C05457=1013.009,-114.708,391.527,-28.818,50.485,-33.096
C05458=1013.004,-115.096,391.557,-28.834,50.637,-33.068
C05459=1013.000,-115.485,391.587,-28.849,50.788,-33.043
C05460=1012.996,-115.873,391.617,-28.865,50.941,-33.016
C05461=1012.993,-116.261,391.647,-28.881,51.094,-32.989
C05462=1012.990,-116.650,391.676,-28.897,51.248,-32.964
C05463=1012.985,-117.038,391.706,-28.913,51.403,-32.938
C05464=1012.982,-117.427,391.737,-28.928,51.558,-32.911
C05465=1012.978,-117.814,391.766,-28.944,51.713,-32.886
C05466=1012.974,-118.203,391.796,-28.960,51.870,-32.860
C05467=1012.970,-118.591,391.826,-28.977,52.028,-32.834
C05468=1012.966,-118.979,391.856,-28.993,52.187,-32.809
C05469=1012.962,-119.367,391.886,-29.009,52.345,-32.783
C05470=1012.959,-119.756,391.916,-29.025,52.504,-32.759
C05471=1012.955,-120.143,391.945,-29.042,52.665,-32.734
C05472=1012.951,-120.532,391.976,-29.058,52.825,-32.709
C05473=1012.947,-120.920,392.005,-29.075,52.986,-32.685
C05474=1012.943,-121.308,392.035,-29.091,53.148,-32.660
C05475=1012.939,-121.696,392.065,-29.108,53.311,-32.636
C05476=1012.936,-122.084,392.095,-29.125,53.475,-32.612
C05477=1012.932,-122.472,392.125,-29.141,53.639,-32.587
C05478=1012.928,-122.861,392.155,-29.158,53.804,-32.564
C05479=1012.924,-123.248,392.184,-29.176,53.969,-32.541
C05480=1012.920,-123.637,392.215,-29.193,54.135,-32.518
C05481=1012.917,-124.025,392.244,-29.210,54.303,-32.495
C05482=1012.913,-124.413,392.274,-29.227,54.470,-32.472
C05483=1012.909,-124.800,392.304,-29.244,54.638,-32.449
C05484=1012.905,-125.188,392.334,-29.262,54.807,-32.427
C05485=1012.901,-125.577,392.364,-29.280,54.977,-32.405
C05486=1012.898,-125.964,392.394,-29.297,55.147,-32.383
C05487=1012.894,-126.352,392.424,-29.315,55.317,-32.362
C05488=1012.890,-126.741,392.454,-29.333,55.489,-32.340
C05489=1012.886,-127.128,392.484,-29.351,55.662,-32.319
C05490=1012.883,-127.516,392.514,-29.369,55.833,-32.297
C05491=1012.878,-127.904,392.544,-29.388,56.007,-32.278
C05492=1012.875,-128.292,392.574,-29.406,56.181,-32.258
C05493=1012.871,-128.679,392.604,-29.424,56.355,-32.238
C05494=1012.867,-129.067,392.634,-29.443,56.531,-32.217
C05495=1012.863,-129.455,392.664,-29.462,56.707,-32.197
C05496=1012.860,-129.843,392.694,-29.481,56.884,-32.179
C05497=1012.855,-130.231,392.724,-29.500,57.062,-32.160
C05498=1012.852,-130.619,392.754,-29.519,57.238,-32.142
C05499=1012.848,-131.006,392.784,-29.538,57.418,-32.123
C05500=1012.845,-131.394,392.814,-29.558,57.597,-32.106
C05501=1012.840,-131.782,392.844,-29.578,57.777,-32.088
C05502=1012.837,-132.170,392.874,-29.597,57.956,-32.071
C05503=1012.833,-132.558,392.903,-29.618,58.138,-32.054
C05504=1012.830,-132.945,392.934,-29.637,58.320,-32.037
C05505=1012.825,-133.333,392.964,-29.658,58.502,-32.021
C05506=1012.822,-133.721,392.994,-29.678,58.685,-32.005
C05507=1012.818,-134.108,393.024,-29.699,58.868,-31.991
C05508=1013.072,-134.133,392.609,-28.595,48.020,-33.821
C05509=1013.077,-133.746,392.579,-28.574,47.825,-33.863
C05510=1013.082,-133.358,392.550,-28.553,47.631,-33.906
C05511=1013.087,-132.970,392.521,-28.532,47.438,-33.948
C05512=1013.092,-132.582,392.491,-28.511,47.244,-33.991
C05513=1013.097,-132.194,392.461,-28.490,47.051,-34.034
C05514=1013.103,-131.806,392.431,-28.469,46.860,-34.077
C05515=1013.108,-131.418,392.402,-28.448,46.669,-34.121
C05516=1013.113,-131.031,392.372,-28.427,46.479,-34.165
C05517=1013.118,-130.643,392.343,-28.406,46.290,-34.208
C05518=1013.122,-130.255,392.314,-28.384,46.101,-34.254
C05519=1013.127,-129.868,392.283,-28.363,45.913,-34.297
C05520=1013.132,-129.480,392.254,-28.342,45.725,-34.342
C05521=1013.138,-129.092,392.225,-28.321,45.538,-34.387
C05522=1013.143,-128.704,392.195,-28.300,45.352,-34.432
C05523=1013.148,-128.316,392.165,-28.279,45.168,-34.477
C05524=1013.153,-127.928,392.136,-28.257,44.983,-34.524
C05525=1013.158,-127.540,392.107,-28.236,44.799,-34.569
C05526=1013.164,-127.152,392.077,-28.215,44.616,-34.614
C05527=1013.168,-126.764,392.047,-28.193,44.434,-34.660
C05528=1013.173,-126.376,392.018,-28.172,44.252,-34.706
C05529=1013.179,-125.988,391.989,-28.151,44.071,-34.753
C05530=1013.183,-125.600,391.959,-28.130,43.891,-34.799
C05531=1013.189,-125.212,391.929,-28.108,43.712,-34.846
C05532=1013.193,-124.825,391.901,-28.087,43.533,-34.893
C05533=1013.199,-124.437,391.871,-28.065,43.355,-34.940
C05534=1013.203,-124.049,391.842,-28.044,43.178,-34.987
C05535=1013.208,-123.661,391.813,-28.023,43.001,-35.034
C05536=1013.214,-123.273,391.783,-28.001,42.826,-35.082
C05537=1013.218,-122.885,391.753,-27.980,42.651,-35.129
C05538=1013.223,-122.497,391.724,-27.958,42.478,-35.176
C05539=1013.229,-122.109,391.695,-27.937,42.304,-35.225
C05540=1013.233,-121.721,391.665,-27.915,42.131,-35.273
C05541=1013.238,-121.333,391.636,-27.894,41.959,-35.320
C05542=1013.244,-120.945,391.606,-27.872,41.788,-35.369
C05543=1013.248,-120.556,391.577,-27.850,41.617,-35.417
C05544=1013.253,-120.168,391.548,-27.829,41.448,-35.464
C05545=1013.259,-119.780,391.518,-27.807,41.280,-35.512
C05546=1013.263,-119.392,391.489,-27.786,41.112,-35.561
C05547=1013.268,-119.004,391.459,-27.764,40.944,-35.610
C05548=1013.274,-118.616,391.430,-27.742,40.778,-35.658
C05549=1013.278,-118.227,391.400,-27.721,40.612,-35.707
C05550=1013.283,-117.839,391.371,-27.699,40.447,-35.756
C05551=1013.287,-117.450,391.342,-27.677,40.283,-35.805
C05552=1013.293,-117.062,391.313,-27.655,40.119,-35.854
C05553=1013.298,-116.674,391.284,-27.634,39.957,-35.902
C05554=1013.302,-116.286,391.254,-27.612,39.795,-35.953
C05555=1013.308,-115.897,391.225,-27.590,39.634,-36.001
C05556=1013.312,-115.508,391.196,-27.568,39.474,-36.051
C05557=1013.318,-115.120,391.166,-27.547,39.314,-36.099
C05558=1013.322,-114.732,391.137,-27.525,39.155,-36.149
C05559=1013.327,-114.344,391.108,-27.503,38.997,-36.198
C05560=1013.332,-113.955,391.078,-27.481,38.840,-36.247
C05561=1013.336,-113.597,391.052,-27.461,38.696,-36.293
C05562=1013.341,-113.179,391.020,-27.438,38.529,-36.346
C05563=1013.346,-112.790,390.991,-27.416,38.374,-36.395
C05564=1013.351,-112.402,390.961,-27.394,38.220,-36.445
C05565=1013.355,-112.013,390.932,-27.372,38.067,-36.494
C05566=1013.361,-111.624,390.903,-27.350,37.914,-36.543
C05567=1013.365,-111.235,390.874,-27.328,37.763,-36.593
C05568=1013.370,-110.847,390.845,-27.306,37.612,-36.642
C05569=1013.374,-110.458,390.815,-27.285,37.462,-36.693
C05570=1013.379,-110.070,390.786,-27.263,37.313,-36.741
C05571=1013.384,-109.681,390.757,-27.241,37.165,-36.790
C05572=1013.389,-109.287,390.727,-27.219,37.015,-36.841
C05573=1013.393,-108.870,390.695,-27.195,36.859,-36.892
C05574=1013.395,-108.651,390.679,-27.183,36.776,-36.921
C05575=1013.398,-108.426,390.662,-27.170,36.692,-36.949
C05576=1013.401,-108.196,390.645,-27.157,36.606,-36.979
C05577=1013.404,-107.964,390.627,-27.144,36.521,-37.008
C05578=1013.406,-107.732,390.610,-27.131,36.434,-37.038
C05579=1013.409,-107.502,390.593,-27.118,36.349,-37.068
C05580=1013.413,-107.275,390.576,-27.105,36.265,-37.097
C05581=1013.414,-107.055,390.560,-27.093,36.184,-37.125
C05582=1013.417,-106.841,390.544,-27.081,36.106,-37.152
C05583=1013.422,-106.434,390.512,-27.058,35.958,-37.202
C05584=1013.426,-106.044,390.483,-27.036,35.816,-37.252
C05585=1013.431,-105.655,390.454,-27.015,35.676,-37.300
C05586=1013.435,-105.266,390.425,-26.993,35.537,-37.350
C05587=1013.440,-104.878,390.396,-26.971,35.400,-37.398
C05588=1013.444,-104.490,390.366,-26.949,35.263,-37.447
C05589=1013.448,-104.103,390.338,-26.928,35.127,-37.495
C05590=1013.453,-103.716,390.309,-26.906,34.992,-37.544
C05591=1013.457,-103.330,390.280,-26.885,34.859,-37.592
C05592=1013.462,-102.944,390.250,-26.863,34.726,-37.640
C05593=1013.465,-102.558,390.222,-26.842,34.594,-37.687
C05594=1013.470,-102.174,390.193,-26.821,34.463,-37.736
C05595=1013.474,-101.791,390.164,-26.799,34.334,-37.783
C05596=1013.478,-101.408,390.135,-26.778,34.205,-37.830
C05597=1013.482,-101.026,390.106,-26.757,34.078,-37.877
C05598=1013.487,-100.645,390.078,-26.736,33.951,-37.924
C05599=1013.491,-100.266,390.049,-26.715,33.826,-37.971
C05600=1013.495,-99.888,390.021,-26.694,33.703,-38.017
C05601=1013.498,-99.510,389.993,-26.674,33.580,-38.063
C05602=1013.502,-99.133,389.965,-26.653,33.459,-38.109
C05603=1013.507,-98.758,389.937,-26.633,33.338,-38.155
C05604=1013.511,-98.381,389.908,-26.612,33.218,-38.200
C05605=1013.515,-98.006,389.880,-26.592,33.100,-38.244
C05606=1013.519,-97.632,389.852,-26.572,32.982,-38.290
C05607=1013.522,-97.256,389.824,-26.551,32.865,-38.335
C05608=1013.526,-96.879,389.795,-26.531,32.749,-38.378
C05609=1013.530,-96.503,389.768,-26.511,32.634,-38.423
C05610=1013.535,-96.126,389.739,-26.491,32.519,-38.467
C05611=1013.538,-95.748,389.711,-26.471,32.404,-38.512
C05612=1013.541,-95.368,389.683,-26.450,32.291,-38.556
C05613=1013.545,-94.988,389.654,-26.430,32.178,-38.600
C05614=1013.549,-94.606,389.625,-26.410,32.065,-38.644
C05615=1013.553,-94.223,389.597,-26.390,31.952,-38.689
C05616=1013.557,-93.840,389.568,-26.370,31.842,-38.733
C05617=1013.561,-93.455,389.539,-26.350,31.730,-38.778
C05618=1013.564,-93.069,389.510,-26.329,31.619,-38.822
C05619=1013.568,-92.682,389.481,-26.310,31.510,-38.865
C05620=1013.572,-92.295,389.452,-26.290,31.401,-38.909
C05621=1013.576,-91.907,389.423,-26.269,31.292,-38.952
C05622=1013.579,-91.519,389.394,-26.249,31.184,-38.996
C05623=1013.583,-91.130,389.364,-26.230,31.077,-39.039
C05624=1013.586,-90.775,389.338,-26.212,30.980,-39.080
C05625=1013.588,-90.507,389.318,-26.198,30.907,-39.108
C05626=1013.591,-90.296,389.302,-26.187,30.850,-39.131
C05627=1013.593,-90.062,389.285,-26.176,30.788,-39.157
C05628=1013.594,-89.812,389.266,-26.163,30.721,-39.183
C05629=1013.597,-89.553,389.246,-26.150,30.652,-39.212
C05630=1013.599,-89.297,389.227,-26.137,30.585,-39.240
C05631=1013.602,-89.055,389.209,-26.125,30.522,-39.266
C05632=1013.603,-88.836,389.193,-26.114,30.464,-39.289
C05633=1013.607,-88.451,389.164,-26.095,30.364,-39.331
C05634=1013.610,-88.074,389.136,-26.077,30.268,-39.370
C05635=1013.614,-87.712,389.109,-26.059,30.175,-39.409
C05636=1013.617,-87.344,389.080,-26.041,30.082,-39.448
C05637=1013.620,-86.968,389.052,-26.023,29.988,-39.486
C05638=1013.623,-86.579,389.024,-26.004,29.891,-39.527
C05639=1013.627,-86.173,388.993,-25.984,29.791,-39.568
C05640=1013.629,-85.949,388.977,-25.974,29.737,-39.591
C05641=1013.631,-85.715,388.958,-25.963,29.679,-39.614
C05642=1013.633,-85.476,388.940,-25.951,29.622,-39.639
C05643=1013.634,-85.237,388.922,-25.940,29.564,-39.663
C05644=1013.637,-85.008,388.905,-25.929,29.510,-39.686
C05645=1013.640,-84.589,388.875,-25.910,29.411,-39.728
C05646=1013.643,-84.197,388.845,-25.891,29.319,-39.766
C05647=1013.646,-83.806,388.815,-25.873,29.228,-39.805
C05648=1013.650,-83.410,388.785,-25.855,29.137,-39.844
C05649=1013.653,-83.013,388.756,-25.837,29.047,-39.882
C05650=1013.656,-82.618,388.726,-25.819,28.957,-39.920
C05651=1013.660,-82.220,388.696,-25.801,28.869,-39.957
C05652=1013.662,-81.821,388.666,-25.783,28.780,-39.996
C05653=1013.665,-81.423,388.636,-25.765,28.694,-40.032
C05654=1013.668,-81.027,388.607,-25.748,28.608,-40.069
C05655=1013.672,-80.629,388.577,-25.731,28.524,-40.105
C05656=1013.674,-80.231,388.547,-25.713,28.439,-40.142
C05657=1013.677,-79.831,388.516,-25.696,28.356,-40.177
C05658=1013.680,-79.431,388.487,-25.679,28.273,-40.214
C05659=1013.683,-79.031,388.456,-25.662,28.192,-40.248
C05660=1013.686,-78.630,388.426,-25.645,28.110,-40.284
C05661=1013.689,-78.228,388.396,-25.629,28.030,-40.318
C05662=1013.692,-77.828,388.366,-25.612,27.951,-40.352
C05663=1013.694,-77.426,388.336,-25.596,27.873,-40.386
C05664=1013.697,-77.024,388.305,-25.579,27.795,-40.421
C05665=1013.700,-76.622,388.275,-25.563,27.718,-40.454
C05666=1013.703,-76.219,388.245,-25.547,27.643,-40.486
C05667=1013.705,-75.817,388.214,-25.531,27.568,-40.519
C05668=1013.708,-75.414,388.183,-25.516,27.493,-40.552
C05669=1013.710,-75.011,388.154,-25.500,27.420,-40.584
C05670=1013.714,-74.608,388.123,-25.485,27.349,-40.615
C05671=1013.715,-74.205,388.093,-25.469,27.277,-40.646
C05672=1013.718,-73.801,388.062,-25.454,27.206,-40.675
C05673=1013.721,-73.398,388.032,-25.440,27.137,-40.706
C05674=1013.723,-72.994,388.001,-25.425,27.068,-40.737
C05675=1013.725,-72.590,387.971,-25.410,27.000,-40.766
C05676=1013.728,-72.186,387.940,-25.396,26.934,-40.795
C05677=1013.731,-71.783,387.910,-25.381,26.868,-40.823
C05678=1013.733,-71.379,387.880,-25.367,26.804,-40.852
C05679=1013.735,-70.975,387.849,-25.353,26.739,-40.879
C05680=1013.737,-70.571,387.818,-25.340,26.676,-40.908
C05681=1013.739,-70.167,387.788,-25.326,26.614,-40.934
C05682=1013.742,-69.762,387.757,-25.313,26.552,-40.961
C05683=1013.744,-69.358,387.727,-25.300,26.492,-40.986
C05684=1013.746,-68.954,387.697,-25.286,26.432,-41.013
C05685=1013.747,-68.549,387.666,-25.274,26.375,-41.038
C05686=1013.750,-68.145,387.636,-25.261,26.316,-41.064
C05687=1013.752,-67.741,387.605,-25.248,26.259,-41.087
C05688=1013.754,-67.338,387.575,-25.236,26.204,-41.111
C05689=1013.755,-66.933,387.544,-25.224,26.149,-41.136
C05690=1013.758,-66.530,387.512,-25.212,26.095,-41.159
C05691=1013.760,-66.127,387.482,-25.200,26.042,-41.180
C05692=1013.762,-65.723,387.452,-25.189,25.990,-41.203
C05693=1013.764,-65.320,387.421,-25.177,25.938,-41.225
C05694=1013.765,-64.918,387.391,-25.166,25.888,-41.247
C05695=1013.767,-64.516,387.360,-25.155,25.839,-41.268
C05696=1013.768,-64.114,387.329,-25.144,25.791,-41.288
C05697=1013.770,-63.712,387.300,-25.134,25.744,-41.308
C05698=1013.772,-63.311,387.269,-25.123,25.697,-41.328
C05699=1013.774,-62.911,387.238,-25.113,25.651,-41.347
C05700=1013.775,-62.510,387.208,-25.103,25.607,-41.366
C05701=1013.777,-62.110,387.177,-25.094,25.563,-41.384
C05702=1013.778,-61.711,387.147,-25.084,25.520,-41.401
C05703=1013.780,-61.312,387.116,-25.075,25.478,-41.418
C05704=1013.782,-60.914,387.086,-25.066,25.437,-41.435
C05705=1013.783,-60.515,387.056,-25.057,25.397,-41.452
C05706=1013.784,-60.119,387.026,-25.048,25.358,-41.467
C05707=1013.786,-59.722,386.996,-25.039,25.320,-41.483
C05708=1013.787,-59.327,386.966,-25.031,25.282,-41.497
C05709=1013.789,-58.930,386.936,-25.023,25.246,-41.512
C05710=1013.790,-58.535,386.906,-25.015,25.211,-41.525
C05711=1013.791,-58.140,386.875,-25.007,25.176,-41.539
C05712=1013.792,-57.746,386.845,-25.000,25.143,-41.552
C05713=1013.794,-57.353,386.815,-24.993,25.110,-41.564
C05714=1013.794,-56.959,386.785,-24.986,25.078,-41.577
C05715=1013.795,-56.566,386.755,-24.979,25.046,-41.587
C05716=1013.796,-56.173,386.725,-24.972,25.016,-41.598
C05717=1013.797,-55.781,386.695,-24.966,24.987,-41.610
C05718=1013.798,-55.388,386.665,-24.959,24.958,-41.620
C05719=1013.799,-54.996,386.635,-24.953,24.931,-41.631
C05720=1013.800,-54.603,386.605,-24.947,24.904,-41.640
C05721=1013.802,-54.211,386.575,-24.942,24.878,-41.647
C05722=1013.802,-53.818,386.545,-24.936,24.853,-41.656
C05723=1013.803,-53.427,386.515,-24.931,24.828,-41.664
C05724=1013.804,-53.034,386.486,-24.926,24.805,-41.672
C05725=1013.804,-52.641,386.455,-24.921,24.781,-41.679
C05726=1013.805,-52.248,386.425,-24.916,24.760,-41.686
C05727=1013.807,-51.856,386.395,-24.912,24.738,-41.693
C05728=1013.807,-51.464,386.366,-24.907,24.718,-41.698
C05729=1013.807,-51.072,386.335,-24.903,24.698,-41.704
C05730=1013.808,-50.679,386.305,-24.899,24.679,-41.708
C05731=1013.809,-50.287,386.275,-24.896,24.662,-41.712
C05732=1013.810,-49.893,386.244,-24.892,24.644,-41.717
C05733=1013.810,-49.501,386.215,-24.889,24.628,-41.720
C05734=1013.810,-49.109,386.184,-24.885,24.612,-41.723
C05735=1013.811,-48.716,386.154,-24.883,24.598,-41.725
C05736=1013.812,-48.324,386.123,-24.880,24.584,-41.728
C05737=1013.811,-47.931,386.094,-24.877,24.571,-41.729
C05738=1013.812,-47.538,386.064,-24.875,24.558,-41.731
C05739=1013.813,-47.146,386.033,-24.873,24.547,-41.731
C05740=1013.813,-46.753,386.003,-24.871,24.536,-41.732
C05741=1013.813,-46.361,385.973,-24.869,24.525,-41.732
C05742=1013.814,-45.968,385.942,-24.867,24.517,-41.731
C05743=1013.814,-45.575,385.912,-24.866,24.508,-41.731
C05744=1013.814,-45.182,385.882,-24.865,24.501,-41.729
C05745=1013.814,-44.789,385.852,-24.864,24.494,-41.727
C05746=1013.814,-44.397,385.821,-24.863,24.489,-41.724
C05747=1013.814,-44.004,385.791,-24.863,24.483,-41.721
C05748=1013.814,-43.611,385.761,-24.862,24.479,-41.719
C05749=1013.814,-43.217,385.730,-24.862,24.475,-41.715
C05750=1013.815,-42.824,385.700,-24.862,24.473,-41.711
C05751=1013.815,-42.431,385.670,-24.862,24.471,-41.706
C05752=1013.814,-42.039,385.640,-24.863,24.469,-41.702
C05753=1013.814,-41.645,385.609,-24.863,24.469,-41.696
C05754=1013.814,-41.253,385.578,-24.864,24.469,-41.690
C05755=1013.814,-40.860,385.548,-24.865,24.471,-41.684
C05756=1013.815,-40.466,385.518,-24.866,24.473,-41.677
C05757=1013.814,-40.073,385.487,-24.868,24.476,-41.670
C05758=1013.814,-39.680,385.457,-24.869,24.479,-41.663
C05759=1013.813,-39.287,385.426,-24.871,24.483,-41.654
C05760=1013.813,-38.894,385.396,-24.873,24.489,-41.645
C05761=1013.813,-38.501,385.365,-24.875,24.495,-41.637
C05762=1013.812,-38.107,385.336,-24.878,24.501,-41.626
C05763=1013.812,-37.713,385.305,-24.880,24.509,-41.618
C05764=1013.812,-37.320,385.275,-24.883,24.518,-41.606
C05765=1013.811,-36.927,385.244,-24.886,24.526,-41.596
C05766=1013.811,-36.533,385.213,-24.889,24.536,-41.586
C05767=1013.810,-36.141,385.182,-24.892,24.547,-41.574
C05768=1013.810,-35.747,385.152,-24.896,24.558,-41.562
C05769=1013.809,-35.354,385.121,-24.899,24.570,-41.550
C05770=1013.809,-34.961,385.090,-24.903,24.583,-41.537
C05771=1013.808,-34.567,385.060,-24.907,24.596,-41.523
C05772=1013.807,-34.174,385.029,-24.912,24.611,-41.509
C05773=1013.807,-33.781,385.000,-24.916,24.626,-41.496
C05774=1013.806,-33.387,384.969,-24.921,24.643,-41.481
C05775=1013.806,-32.994,384.938,-24.925,24.659,-41.466
C05776=1013.804,-32.601,384.908,-24.930,24.676,-41.451
C05777=1013.804,-32.207,384.877,-24.935,24.695,-41.435
C05778=1013.803,-31.814,384.846,-24.941,24.714,-41.419
C05779=1013.802,-31.420,384.814,-24.946,24.734,-41.402
C05780=1013.800,-31.027,384.785,-24.952,24.755,-41.385
C05781=1013.800,-30.633,384.754,-24.958,24.776,-41.367
C05782=1013.799,-30.240,384.723,-24.964,24.798,-41.350
C05783=1013.798,-29.847,384.693,-24.970,24.821,-41.332
C05784=1013.797,-29.454,384.662,-24.977,24.845,-41.313
C05785=1013.796,-29.061,384.631,-24.983,24.869,-41.294
C05786=1013.795,-28.667,384.600,-24.990,24.894,-41.274
C05787=1013.794,-28.275,384.569,-24.996,24.920,-41.255
C05788=1013.793,-27.880,384.539,-25.004,24.947,-41.234
C05789=1013.791,-27.487,384.508,-25.011,24.975,-41.214
C05790=1013.790,-27.094,384.477,-25.018,25.003,-41.193
C05791=1013.789,-26.701,384.447,-25.026,25.032,-41.171
C05792=1013.788,-26.307,384.415,-25.034,25.062,-41.149
C05793=1013.787,-25.915,384.385,-25.041,25.092,-41.128
C05794=1013.786,-25.522,384.354,-25.050,25.123,-41.105
C05795=1013.784,-25.128,384.323,-25.058,25.155,-41.082
C05796=1013.783,-24.735,384.293,-25.066,25.188,-41.058
C05797=1013.781,-24.342,384.261,-25.075,25.222,-41.035
C05798=1013.781,-23.949,384.231,-25.083,25.255,-41.010
C05799=1013.779,-23.556,384.200,-25.092,25.291,-40.986
C05800=1013.777,-23.163,384.168,-25.101,25.327,-40.962
C05801=1013.775,-22.770,384.139,-25.110,25.363,-40.937
C05802=1013.774,-22.376,384.107,-25.120,25.400,-40.912
C05803=1013.773,-21.983,384.077,-25.129,25.438,-40.885
C05804=1013.771,-21.590,384.046,-25.139,25.477,-40.859
C05805=1013.769,-21.197,384.015,-25.149,25.517,-40.832
C05806=1013.768,-20.804,383.984,-25.159,25.557,-40.805
C05807=1013.766,-20.407,383.953,-25.169,25.598,-40.777
C05808=1013.764,-20.058,383.925,-25.178,25.635,-40.753
C05809=1013.763,-19.852,383.909,-25.183,25.657,-40.738
C05810=1013.762,-19.621,383.891,-25.189,25.683,-40.721
C05811=1013.761,-19.365,383.871,-25.196,25.711,-40.702
C05812=1013.760,-19.091,383.849,-25.204,25.741,-40.683
C05813=1013.759,-18.812,383.828,-25.211,25.772,-40.663
C05814=1013.757,-18.540,383.805,-25.219,25.803,-40.642
C05815=1013.757,-18.287,383.786,-25.226,25.832,-40.623
C05816=1013.756,-18.060,383.768,-25.232,25.858,-40.607
C05817=1013.753,-17.664,383.737,-25.243,25.905,-40.577
C05818=1013.751,-17.275,383.706,-25.254,25.951,-40.547
C05819=1013.749,-16.877,383.674,-25.266,26.000,-40.516
C05820=1013.747,-16.481,383.643,-25.278,26.049,-40.485
C05821=1013.745,-16.085,383.612,-25.289,26.098,-40.454
C05822=1013.744,-15.690,383.581,-25.301,26.148,-40.423
C05823=1013.742,-15.303,383.551,-25.312,26.197,-40.392
C05824=1013.739,-14.923,383.520,-25.324,26.248,-40.360
C05825=1013.737,-14.548,383.491,-25.336,26.296,-40.329
C05826=1013.735,-14.173,383.461,-25.348,26.348,-40.297
C05827=1013.733,-13.792,383.431,-25.360,26.399,-40.264
C05828=1013.732,-13.399,383.400,-25.372,26.453,-40.232
C05829=1013.729,-12.995,383.368,-25.385,26.510,-40.198
C05830=1013.726,-12.584,383.336,-25.398,26.568,-40.162
C05831=1013.724,-12.170,383.303,-25.412,26.627,-40.126
C05832=1013.722,-11.755,383.271,-25.426,26.688,-40.089
C05833=1013.719,-11.337,383.238,-25.440,26.750,-40.052
C05834=1013.717,-10.919,383.204,-25.454,26.812,-40.014
C05835=1013.714,-10.500,383.171,-25.468,26.876,-39.977
C05836=1013.712,-10.080,383.138,-25.483,26.940,-39.938
C05837=1013.709,-9.658,383.105,-25.497,27.005,-39.900
C05838=1013.707,-9.236,383.071,-25.512,27.072,-39.860
C05839=1013.704,-8.814,383.038,-25.527,27.139,-39.821
C05840=1013.702,-8.603,383.021,-25.534,27.173,-39.800
C05841=1013.701,-8.392,383.004,-25.542,27.207,-39.781
C05842=1013.699,-8.034,382.976,-25.555,27.266,-39.747
C05843=1013.696,-7.755,382.954,-25.565,27.311,-39.721
C05844=1013.696,-7.541,382.937,-25.572,27.347,-39.701
C05845=1013.694,-7.327,382.920,-25.580,27.383,-39.679
C05846=1013.693,-7.112,382.903,-25.588,27.418,-39.659
C05847=1013.692,-6.897,382.885,-25.596,27.455,-39.638
C05848=1013.690,-6.680,382.868,-25.604,27.493,-39.617
C05849=1013.688,-6.465,382.852,-25.612,27.529,-39.595
C05850=1013.687,-6.248,382.834,-25.620,27.566,-39.574
C05851=1013.686,-6.031,382.816,-25.628,27.604,-39.553
C05852=1013.684,-5.815,382.800,-25.636,27.641,-39.532
C05853=1013.682,-5.598,382.783,-25.644,27.679,-39.510
C05854=1013.681,-5.384,382.766,-25.652,27.717,-39.489
C05855=1013.679,-4.969,382.733,-25.668,27.790,-39.448
C05856=1013.675,-4.579,382.702,-25.683,27.860,-39.408
C05857=1013.673,-4.199,382.671,-25.697,27.929,-39.370
C05858=1013.669,-3.815,382.641,-25.712,27.999,-39.329
C05859=1013.667,-3.413,382.609,-25.727,28.074,-39.289
C05860=1013.664,-3.001,382.577,-25.743,28.150,-39.247
C05861=1013.661,-2.591,382.544,-25.759,28.227,-39.204
C05862=1013.658,-2.183,382.512,-25.776,28.305,-39.161
C05863=1013.655,-1.777,382.479,-25.791,28.382,-39.119
C05864=1013.651,-1.373,382.447,-25.807,28.461,-39.076
C05865=1013.648,-0.970,382.415,-25.824,28.540,-39.033
C05866=1013.645,-0.570,382.384,-25.840,28.619,-38.991
C05867=1013.642,-0.172,382.352,-25.856,28.698,-38.948
C05868=1013.639,0.223,382.320,-25.872,28.778,-38.906
C05869=1013.636,0.617,382.289,-25.888,28.858,-38.862
C05870=1013.633,1.012,382.258,-25.904,28.940,-38.819
C05871=1013.629,1.410,382.226,-25.920,29.021,-38.776
C05872=1013.627,1.801,382.195,-25.936,29.103,-38.734
C05873=1013.623,2.173,382.166,-25.952,29.181,-38.693
C05874=1013.620,2.515,382.138,-25.966,29.253,-38.655
C05875=1013.618,2.838,382.112,-25.979,29.322,-38.618
C05876=1013.615,3.162,382.087,-25.993,29.392,-38.581
C05877=1013.612,3.506,382.060,-26.007,29.466,-38.544
C05878=1013.609,3.878,382.030,-26.023,29.548,-38.501
C05879=1013.606,4.269,381.999,-26.039,29.634,-38.457
C05880=1013.603,4.658,381.968,-26.056,29.719,-38.413
C05881=1013.599,5.047,381.937,-26.072,29.807,-38.368
C05882=1013.595,5.437,381.906,-26.089,29.894,-38.324
C05883=1013.593,5.829,381.874,-26.106,29.983,-38.280
C05884=1013.589,6.222,381.843,-26.122,30.072,-38.235
C05885=1013.586,6.613,381.813,-26.139,30.163,-38.188
C05886=1013.582,6.999,381.782,-26.156,30.252,-38.145
C05887=1013.578,7.379,381.751,-26.172,30.341,-38.100
C05888=1013.575,7.758,381.721,-26.188,30.430,-38.056
C05889=1013.572,8.133,381.690,-26.205,30.520,-38.011
C05890=1013.568,8.508,381.661,-26.221,30.609,-37.968
C05891=1013.565,8.881,381.631,-26.237,30.698,-37.923
C05892=1013.562,9.254,381.602,-26.254,30.789,-37.879
C05893=1013.558,9.629,381.572,-26.270,30.881,-37.835
C05894=1013.555,10.004,381.542,-26.287,30.973,-37.791
C05895=1013.551,10.383,381.512,-26.303,31.066,-37.746
C05896=1013.548,10.756,381.482,-26.319,31.159,-37.701
C05897=1013.544,11.121,381.453,-26.335,31.250,-37.658
C05898=1013.540,11.485,381.424,-26.352,31.342,-37.613
C05899=1013.536,11.856,381.394,-26.368,31.436,-37.569
C05900=1013.533,12.238,381.364,-26.385,31.534,-37.522
C05901=1013.530,12.622,381.333,-26.402,31.633,-37.476
C05902=1013.526,13.006,381.302,-26.419,31.732,-37.430
C05903=1013.522,13.389,381.272,-26.436,31.831,-37.384
C05904=1013.518,13.770,381.242,-26.453,31.932,-37.337
C05905=1013.514,14.151,381.211,-26.470,32.032,-37.290
C05906=1013.511,14.531,381.181,-26.487,32.133,-37.244
C05907=1013.507,14.911,381.151,-26.504,32.235,-37.198
C05908=1013.503,15.291,381.121,-26.521,32.336,-37.151
C05909=1013.499,15.671,381.090,-26.538,32.439,-37.104
C05910=1013.495,16.053,381.060,-26.555,32.543,-37.056
C05911=1013.491,16.435,381.029,-26.572,32.648,-37.010
C05912=1013.487,16.819,380.998,-26.589,32.754,-36.962
C05913=1013.482,17.205,380.968,-26.606,32.860,-36.915
C05914=1013.479,17.592,380.937,-26.624,32.969,-36.866
C05915=1013.475,17.983,380.906,-26.641,33.078,-36.818
C05916=1013.471,18.373,380.875,-26.659,33.188,-36.770
C05917=1013.466,18.774,380.843,-26.677,33.302,-36.719
C05918=1013.462,19.175,380.811,-26.695,33.417,-36.670
C05919=1013.460,19.379,380.795,-26.704,33.475,-36.645
C05920=1013.458,19.600,380.777,-26.714,33.539,-36.617
C05921=1013.455,19.842,380.758,-26.725,33.609,-36.586
C05922=1013.452,20.102,380.737,-26.736,33.684,-36.554
C05923=1013.449,20.372,380.716,-26.748,33.763,-36.520
C05924=1013.447,20.640,380.694,-26.760,33.841,-36.487
C05925=1013.443,20.900,380.673,-26.772,33.918,-36.454
C05926=1013.441,21.148,380.653,-26.783,33.991,-36.423
C05927=1013.438,21.376,380.636,-26.793,34.058,-36.394
C05928=1013.434,21.764,380.605,-26.811,34.173,-36.346
C05929=1013.431,22.092,380.579,-26.826,34.271,-36.304
C05930=1013.427,22.423,380.552,-26.840,34.370,-36.263
C05931=1013.424,22.700,380.530,-26.853,34.454,-36.228
C05932=1013.420,23.064,380.501,-26.869,34.564,-36.182
C05933=1013.415,23.479,380.468,-26.888,34.690,-36.129
C05934=1013.411,23.820,380.441,-26.903,34.793,-36.087
C05935=1013.407,24.199,380.411,-26.920,34.910,-36.039
C05936=1013.403,24.594,380.379,-26.937,35.032,-35.989
C05937=1013.398,24.990,380.348,-26.955,35.155,-35.940
C05938=1013.394,25.386,380.316,-26.973,35.278,-35.889
C05939=1013.389,25.784,380.285,-26.990,35.403,-35.839
C05940=1013.385,26.182,380.253,-27.008,35.529,-35.789
C05941=1013.380,26.578,380.222,-27.026,35.653,-35.739
C05942=1013.375,26.972,380.190,-27.043,35.779,-35.689
C05943=1013.371,27.366,380.159,-27.060,35.904,-35.640
C05944=1013.366,27.758,380.127,-27.078,36.030,-35.590
C05945=1013.362,28.151,380.096,-27.095,36.157,-35.541
C05946=1013.357,28.544,380.065,-27.112,36.284,-35.492
C05947=1013.352,28.940,380.034,-27.130,36.412,-35.442
C05948=1013.348,29.335,380.002,-27.147,36.542,-35.392
C05949=1013.343,29.730,379.971,-27.164,36.672,-35.342
C05950=1013.339,30.125,379.939,-27.181,36.802,-35.293
C05951=1013.334,30.520,379.907,-27.199,36.933,-35.243
C05952=1013.329,30.915,379.876,-27.216,37.066,-35.194
C05953=1013.324,31.311,379.845,-27.233,37.197,-35.145
C05954=1013.320,31.706,379.813,-27.250,37.329,-35.095
C05955=1013.315,32.101,379.782,-27.267,37.463,-35.045
C05956=1013.309,32.496,379.751,-27.284,37.597,-34.996
C05957=1013.305,32.891,379.719,-27.301,37.732,-34.947
C05958=1013.300,33.286,379.688,-27.318,37.867,-34.897
C05959=1013.295,33.681,379.656,-27.335,38.003,-34.848
C05960=1013.290,34.077,379.625,-27.352,38.139,-34.800
C05961=1013.286,34.472,379.594,-27.369,38.276,-34.750
C05962=1013.281,34.867,379.562,-27.386,38.413,-34.702
C05963=1013.276,35.262,379.531,-27.402,38.551,-34.653
C05964=1013.271,35.658,379.499,-27.419,38.690,-34.604
C05965=1013.266,36.054,379.469,-27.436,38.829,-34.555
C05966=1013.261,36.448,379.438,-27.452,38.969,-34.506
C05967=1013.256,36.843,379.406,-27.469,39.109,-34.457
C05968=1013.251,37.239,379.374,-27.485,39.250,-34.409
C05969=1013.246,37.634,379.343,-27.502,39.391,-34.361
C05970=1013.241,38.030,379.311,-27.518,39.533,-34.312
C05971=1013.237,38.425,379.280,-27.535,39.676,-34.264
C05972=1013.231,38.821,379.249,-27.551,39.820,-34.216
C05973=1013.227,39.216,379.218,-27.567,39.964,-34.168
C05974=1013.221,39.611,379.186,-27.584,40.108,-34.121
C05975=1013.216,40.006,379.155,-27.600,40.252,-34.072
C05976=1013.211,40.402,379.124,-27.616,40.398,-34.024
C05977=1013.206,40.797,379.093,-27.632,40.544,-33.977
C05978=1013.201,41.192,379.061,-27.648,40.690,-33.930
C05979=1013.196,41.588,379.029,-27.664,40.838,-33.881
C05980=1013.191,41.984,378.998,-27.680,40.985,-33.835
C05981=1013.185,42.378,378.967,-27.696,41.134,-33.788
C05982=1013.180,42.774,378.937,-27.712,41.282,-33.741
C05983=1013.175,43.170,378.905,-27.728,41.431,-33.694
C05984=1013.170,43.565,378.873,-27.743,41.581,-33.647
C05985=1013.165,43.961,378.843,-27.759,41.732,-33.600
C05986=1013.160,44.357,378.811,-27.775,41.883,-33.553
C05987=1013.155,44.752,378.780,-27.790,42.035,-33.507
C05988=1013.150,45.148,378.748,-27.806,42.186,-33.461
C05989=1013.144,45.543,378.716,-27.821,42.339,-33.414
C05990=1013.139,45.939,378.686,-27.837,42.492,-33.369
C05991=1013.134,46.334,378.655,-27.852,42.646,-33.323
C05992=1013.128,46.730,378.623,-27.868,42.800,-33.278
C05993=1013.123,47.125,378.592,-27.883,42.955,-33.231
C05994=1013.118,47.521,378.561,-27.898,43.109,-33.186
C05995=1013.112,47.917,378.530,-27.913,43.266,-33.141
C05996=1013.108,48.313,378.499,-27.929,43.423,-33.096
C05997=1013.103,48.708,378.468,-27.944,43.579,-33.051
C05998=1013.097,49.104,378.436,-27.959,43.736,-33.007
C05999=1013.092,49.500,378.405,-27.974,43.893,-32.963
C06000=1013.086,49.896,378.374,-27.988,44.052,-32.918
C06001=1013.082,50.291,378.342,-28.003,44.211,-32.874
C06002=1013.076,50.687,378.312,-28.018,44.371,-32.830
C06003=1013.070,51.083,378.281,-28.033,44.530,-32.786
C06004=1013.065,51.478,378.249,-28.048,44.692,-32.742
C06005=1013.060,51.874,378.218,-28.062,44.852,-32.699
C06006=1013.055,52.270,378.187,-28.077,45.014,-32.655
C06007=1013.049,52.666,378.156,-28.092,45.176,-32.612
C06008=1013.044,53.062,378.125,-28.106,45.338,-32.569
C06009=1013.039,53.457,378.094,-28.121,45.501,-32.527
C06010=1013.033,53.854,378.063,-28.135,45.665,-32.484
C06011=1013.028,54.249,378.032,-28.150,45.829,-32.441
C06012=1013.022,54.646,378.001,-28.164,45.994,-32.399
C06013=1013.018,55.041,377.969,-28.178,46.159,-32.358
C06014=1013.012,55.437,377.938,-28.193,46.324,-32.316
C06015=1013.007,55.833,377.907,-28.207,46.490,-32.275
C06016=1013.001,56.229,377.876,-28.221,46.656,-32.233
C06017=1012.996,56.625,377.845,-28.235,46.824,-32.192
C06018=1012.991,57.021,377.814,-28.249,46.991,-32.151
C06019=1012.985,57.417,377.783,-28.263,47.159,-32.111
C06020=1012.980,57.812,377.752,-28.277,47.327,-32.071
C06021=1012.974,58.209,377.720,-28.291,47.497,-32.030
C06022=1012.969,58.605,377.690,-28.305,47.665,-31.991
C06023=1012.964,59.001,377.658,-28.319,47.836,-31.951
C06024=1012.958,59.397,377.628,-28.333,48.006,-31.912
C06025=1012.952,59.792,377.597,-28.347,48.177,-31.873
C06026=1012.947,60.188,377.566,-28.361,48.349,-31.833
C06027=1012.942,60.584,377.535,-28.375,48.520,-31.795
C06028=1012.936,60.980,377.504,-28.388,48.691,-31.757
C06029=1012.931,61.376,377.473,-28.402,48.864,-31.719
C06030=1012.925,61.772,377.442,-28.416,49.037,-31.681
C06031=1012.920,62.170,377.411,-28.429,49.211,-31.643
C06032=1012.917,62.453,377.389,-28.439,49.335,-31.616
C06033=1012.913,62.673,377.372,-28.447,49.431,-31.596
C06034=1012.910,62.915,377.353,-28.455,49.537,-31.574
C06035=1012.906,63.164,377.333,-28.463,49.646,-31.550
C06036=1012.904,63.398,377.315,-28.472,49.750,-31.528
C06037=1012.901,63.610,377.298,-28.479,49.843,-31.508
C06038=1012.898,64.015,377.262,-28.483,49.898,-31.495
C06039=1012.898,64.234,377.242,-28.483,49.903,-31.493
C06040=1012.898,64.461,377.221,-28.483,49.908,-31.490
C06041=1012.896,64.687,377.200,-28.483,49.914,-31.487
C06042=1012.896,64.909,377.178,-28.483,49.919,-31.485
C06043=1012.895,65.128,377.158,-28.483,49.925,-31.481
C06044=1012.894,65.343,377.139,-28.484,49.930,-31.479
C06045=1012.893,65.551,377.119,-28.484,49.936,-31.476
C06046=1012.893,65.944,377.081,-28.484,49.945,-31.471
C06047=1012.891,66.271,377.051,-28.484,49.954,-31.468
C06048=1012.890,66.635,377.017,-28.485,49.963,-31.463
C06049=1012.889,67.033,376.979,-28.485,49.972,-31.458
C06050=1012.888,67.431,376.943,-28.485,49.983,-31.452
C06051=1012.886,67.831,376.905,-28.485,49.993,-31.448
C06052=1012.885,68.243,376.867,-28.486,50.004,-31.442
C06053=1012.884,68.660,376.827,-28.486,50.014,-31.437
C06054=1012.882,69.077,376.788,-28.487,50.025,-31.433
C06055=1012.881,69.483,376.750,-28.487,50.035,-31.427
C06056=1012.880,69.888,376.711,-28.487,50.046,-31.422
C06057=1012.878,70.292,376.674,-28.487,50.056,-31.417
C06058=1012.877,70.697,376.636,-28.488,50.067,-31.412
C06059=1012.876,71.101,376.598,-28.488,50.078,-31.406
C06060=1012.874,71.506,376.560,-28.488,50.088,-31.402
C06061=1012.874,71.911,376.521,-28.489,50.099,-31.397
C06062=1012.872,72.317,376.483,-28.489,50.110,-31.391
C06063=1012.871,72.725,376.445,-28.490,50.120,-31.387
C06064=1012.869,73.134,376.406,-28.490,50.131,-31.382
C06065=1012.868,73.546,376.366,-28.490,50.142,-31.376
C06066=1012.867,73.961,376.327,-28.490,50.152,-31.371
C06067=1012.866,74.180,376.307,-28.491,50.159,-31.368
C06068=1012.865,74.408,376.286,-28.491,50.164,-31.366
C06069=1012.864,74.634,376.264,-28.491,50.171,-31.363
C06070=1012.863,74.849,376.243,-28.491,50.177,-31.360
C06071=1012.863,75.058,376.223,-28.492,50.182,-31.358
C06072=1012.861,75.473,376.185,-28.492,50.193,-31.352
C06073=1012.861,75.882,376.146,-28.492,50.205,-31.348
C06074=1012.859,76.283,376.107,-28.493,50.216,-31.342
C06075=1012.858,76.677,376.070,-28.493,50.226,-31.338
C06076=1012.856,77.064,376.034,-28.493,50.237,-31.333
C06077=1012.855,77.445,375.998,-28.494,50.247,-31.329
C06078=1012.854,77.827,375.961,-28.494,50.258,-31.323
C06079=1012.852,78.211,375.925,-28.494,50.268,-31.319
C06080=1012.850,78.600,375.888,-28.495,50.279,-31.314
C06081=1012.849,78.994,375.850,-28.495,50.290,-31.308
C06082=1012.848,79.396,375.811,-28.495,50.300,-31.304
C06083=1012.846,79.806,375.773,-28.496,50.311,-31.299
C06084=1012.845,80.218,375.734,-28.496,50.322,-31.294
C06085=1012.844,80.600,375.697,-28.497,50.334,-31.289
C06086=1012.842,80.963,375.663,-28.497,50.343,-31.284
C06087=1012.841,81.357,375.625,-28.497,50.355,-31.280
C06088=1012.840,81.772,375.586,-28.498,50.366,-31.274
C06089=1012.838,82.185,375.546,-28.498,50.378,-31.269
C06090=1012.837,82.599,375.507,-28.499,50.390,-31.265
C06091=1012.835,83.010,375.467,-28.499,50.401,-31.260
C06092=1012.834,83.421,375.428,-28.499,50.412,-31.254
C06093=1012.832,83.830,375.389,-28.500,50.425,-31.248
C06094=1012.831,84.239,375.350,-28.500,50.437,-31.244
C06095=1012.829,84.646,375.311,-28.501,50.449,-31.239
C06096=1012.828,85.051,375.272,-28.501,50.460,-31.234
C06097=1012.826,85.455,375.233,-28.501,50.471,-31.229
C06098=1012.825,85.859,375.195,-28.502,50.483,-31.224
C06099=1012.824,86.261,375.156,-28.502,50.495,-31.219
C06100=1012.822,86.661,375.117,-28.503,50.507,-31.214
C06101=1012.821,87.060,375.080,-28.503,50.518,-31.210
C06102=1012.820,87.454,375.041,-28.504,50.529,-31.204
C06103=1012.817,87.839,375.005,-28.504,50.541,-31.200
C06104=1012.816,88.216,374.968,-28.505,50.552,-31.196
C06105=1012.815,88.591,374.932,-28.505,50.563,-31.191
C06106=1012.814,88.969,374.896,-28.505,50.575,-31.186
C06107=1012.812,89.354,374.859,-28.506,50.586,-31.181
C06108=1012.810,89.749,374.820,-28.506,50.597,-31.176
C06109=1012.809,89.984,374.798,-28.506,50.604,-31.173
C06110=1012.809,90.259,374.771,-28.507,50.611,-31.170
C06111=1012.808,90.538,374.745,-28.507,50.618,-31.168
C06112=1012.806,90.784,374.720,-28.507,50.626,-31.164
C06113=1012.805,91.187,374.682,-28.508,50.638,-31.160
C06114=1012.804,91.582,374.645,-28.508,50.650,-31.155
C06115=1012.802,91.976,374.605,-28.509,50.663,-31.149
C06116=1012.801,92.371,374.568,-28.509,50.676,-31.145
C06117=1012.800,92.765,374.530,-28.510,50.687,-31.141
C06118=1012.798,93.160,374.492,-28.510,50.700,-31.135
C06119=1012.797,93.554,374.453,-28.511,50.710,-31.131
C06120=1012.795,93.949,374.415,-28.511,50.722,-31.126
C06121=1012.793,94.344,374.377,-28.511,50.732,-31.122
C06122=1012.792,94.737,374.339,-28.512,50.744,-31.117
C06123=1012.790,95.132,374.300,-28.512,50.756,-31.112
C06124=1012.789,95.527,374.263,-28.513,50.769,-31.107
C06125=1012.787,95.921,374.224,-28.513,50.782,-31.103
C06126=1012.786,96.316,374.186,-28.514,50.795,-31.098
C06127=1012.785,96.711,374.148,-28.514,50.809,-31.092
C06128=1012.783,97.105,374.109,-28.515,50.819,-31.088
C06129=1012.781,97.499,374.072,-28.515,50.830,-31.083
C06130=1012.779,97.893,374.032,-28.516,50.842,-31.079
C06131=1012.778,98.288,373.995,-28.516,50.854,-31.074
C06132=1012.776,98.682,373.956,-28.517,50.867,-31.069
C06133=1012.775,99.077,373.918,-28.517,50.880,-31.065
C06134=1012.773,99.471,373.879,-28.518,50.894,-31.060
C06135=1012.772,99.865,373.841,-28.518,50.908,-31.054
C06136=1012.770,100.260,373.802,-28.519,50.918,-31.050
C06137=1012.769,100.654,373.764,-28.519,50.930,-31.046
C06138=1012.767,101.049,373.725,-28.520,50.941,-31.041
C06139=1012.766,101.443,373.687,-28.520,50.954,-31.037
C06140=1012.764,101.838,373.649,-28.521,50.967,-31.032
C06141=1012.763,102.231,373.610,-28.521,50.981,-31.026
C06142=1012.761,102.626,373.572,-28.522,50.994,-31.022
C06143=1012.760,103.020,373.534,-28.523,51.009,-31.016
C06144=1012.758,103.414,373.494,-28.523,51.020,-31.013
C06145=1012.756,103.809,373.455,-28.524,51.031,-31.008
C06146=1012.754,104.202,373.418,-28.524,51.044,-31.004
C06147=1012.753,104.597,373.379,-28.525,51.056,-30.999
C06148=1012.752,104.991,373.340,-28.525,51.069,-30.994
C06149=1012.750,105.386,373.302,-28.526,51.083,-30.989
C06150=1012.748,105.780,373.263,-28.526,51.097,-30.984
C06151=1012.747,106.173,373.225,-28.527,51.111,-30.979
C06152=1012.745,106.568,373.186,-28.528,51.124,-30.975
C06153=1012.743,106.962,373.147,-28.528,51.136,-30.971
C06154=1012.742,107.357,373.109,-28.528,51.147,-30.966
C06155=1012.740,107.751,373.070,-28.529,51.160,-30.962
C06156=1012.738,108.145,373.031,-28.529,51.174,-30.956
C06157=1012.737,108.539,372.993,-28.530,51.187,-30.953
C06158=1012.735,108.933,372.954,-28.531,51.200,-30.948
C06159=1012.734,109.327,372.914,-28.531,51.215,-30.943
C06160=1012.733,109.722,372.876,-28.532,51.229,-30.939
C06161=1012.731,110.115,372.837,-28.533,51.241,-30.934
C06162=1012.729,110.510,372.799,-28.533,51.253,-30.930
C06163=1012.727,110.904,372.760,-28.534,51.267,-30.924
C06164=1012.726,111.298,372.721,-28.534,51.279,-30.920
C06165=1012.724,111.693,372.682,-28.535,51.293,-30.915
C06166=1012.723,112.087,372.643,-28.535,51.307,-30.910
C06167=1012.720,112.481,372.604,-28.536,51.321,-30.906
C06168=1012.719,112.875,372.566,-28.537,51.337,-30.902
C06169=1012.718,113.269,372.527,-28.537,51.348,-30.897
C06170=1012.716,113.664,372.488,-28.538,51.361,-30.893
C06171=1012.714,114.058,372.449,-28.538,51.374,-30.888
C06172=1012.713,114.452,372.410,-28.539,51.387,-30.884
C06173=1012.710,114.846,372.371,-28.540,51.401,-30.879
C06174=1012.710,115.239,372.332,-28.540,51.416,-30.875
C06175=1012.708,115.634,372.293,-28.541,51.430,-30.870
C06176=1012.706,116.028,372.253,-28.542,51.446,-30.865
C06177=1012.705,116.422,372.214,-28.542,51.458,-30.861
C06178=1012.703,116.817,372.175,-28.543,51.471,-30.857
C06179=1012.701,117.211,372.136,-28.543,51.485,-30.851
C06180=1012.699,117.605,372.098,-28.544,51.498,-30.848
C06181=1012.697,117.999,372.058,-28.545,51.511,-30.843
C06182=1012.696,118.393,372.019,-28.545,51.526,-30.838
C06183=1012.694,118.787,371.980,-28.546,51.541,-30.834
C06184=1012.693,119.181,371.940,-28.547,51.556,-30.828
C06185=1012.691,119.576,371.901,-28.547,51.571,-30.824
C06186=1012.690,119.970,371.863,-28.548,51.584,-30.820
C06187=1012.688,120.364,371.824,-28.549,51.596,-30.816
C06188=1012.687,120.758,371.784,-28.549,51.610,-30.811
C06189=1012.684,121.152,371.745,-28.550,51.624,-30.806
C06190=1012.682,121.546,371.706,-28.550,51.638,-30.802
C06191=1012.681,121.940,371.667,-28.551,51.653,-30.798
C06192=1012.679,122.335,371.627,-28.552,51.669,-30.794
C06193=1012.678,122.728,371.588,-28.553,51.685,-30.789
C06194=1012.676,123.123,371.549,-28.553,51.697,-30.785
C06195=1012.674,123.517,371.509,-28.554,51.710,-30.781
C06196=1012.673,123.911,371.470,-28.554,51.724,-30.776
C06197=1012.671,124.305,371.431,-28.555,51.738,-30.771
C06198=1012.669,124.700,371.392,-28.556,51.753,-30.767
C06199=1012.668,125.093,371.352,-28.557,51.768,-30.763
C06200=1012.666,125.488,371.313,-28.557,51.784,-30.758
C06201=1012.665,125.882,371.274,-28.558,51.799,-30.754
C06202=1012.662,126.277,371.234,-28.559,51.813,-30.749
C06203=1012.661,126.670,371.194,-28.559,51.826,-30.745
C06204=1012.659,127.065,371.155,-28.560,51.840,-30.741
C06205=1012.658,127.458,371.115,-28.561,51.854,-30.736
C06206=1012.656,127.853,371.076,-28.561,51.869,-30.732
C06207=1012.654,128.247,371.036,-28.562,51.885,-30.728
C06208=1012.652,128.641,370.997,-28.563,51.900,-30.723
C06209=1012.651,129.035,370.958,-28.564,51.916,-30.719
C06210=1012.650,129.430,370.918,-28.564,51.932,-30.714
C06211=1012.648,129.825,370.878,-28.565,51.944,-30.710
C06212=1012.646,130.219,370.839,-28.566,51.958,-30.705
C06213=1012.645,130.613,370.799,-28.566,51.973,-30.701
C06214=1012.643,131.007,370.760,-28.567,51.988,-30.697
C06215=1012.641,131.401,370.719,-28.568,52.003,-30.693
C06216=1012.639,131.795,370.680,-28.569,52.018,-30.689
C06217=1012.638,132.190,370.641,-28.570,52.035,-30.684
C06218=1012.636,132.584,370.600,-28.570,52.051,-30.679
C06219=1012.634,132.979,370.561,-28.571,52.064,-30.676
C06220=1012.633,133.372,370.522,-28.572,52.079,-30.671
C06221=1012.630,133.767,370.482,-28.572,52.094,-30.668
C06222=1012.630,134.162,370.442,-28.573,52.108,-30.663
C06223=1012.627,134.556,370.402,-28.574,52.124,-30.658
C06224=1012.627,134.786,370.379,-28.574,52.133,-30.655
C06225=1012.626,135.046,370.353,-28.575,52.143,-30.653
C06226=1012.624,135.457,370.311,-28.576,52.161,-30.649
C06227=1012.622,135.825,370.274,-28.577,52.175,-30.645
C06228=1012.620,136.166,370.240,-28.577,52.189,-30.640
C06229=1012.620,136.487,370.207,-28.578,52.201,-30.638
C06230=1012.618,136.807,370.175,-28.578,52.214,-30.634
C06231=1012.616,137.151,370.140,-28.579,52.227,-30.631
C06232=1012.615,137.499,370.105,-28.580,52.241,-30.627
C06233=1012.614,137.800,370.074,-28.581,52.253,-30.624
C06234=1012.612,138.195,370.034,-28.581,52.268,-30.620
C06235=1012.611,138.415,370.012,-28.582,52.277,-30.616
C06236=1012.610,138.650,369.989,-28.582,52.286,-30.614
C06237=1012.609,138.899,369.963,-28.583,52.296,-30.612
C06238=1012.608,139.156,369.937,-28.583,52.306,-30.608
C06239=1012.607,139.419,369.910,-28.584,52.316,-30.606
C06240=1012.606,139.680,369.884,-28.584,52.327,-30.603
C06241=1012.605,139.933,369.858,-28.585,52.337,-30.601
C06242=1012.603,140.176,369.834,-28.585,52.346,-30.598
C06243=1012.602,140.402,369.811,-28.586,52.356,-30.596
C06244=1012.602,140.614,369.789,-28.586,52.363,-30.594
C06245=1012.601,140.831,369.768,-28.587,52.372,-30.591
C06246=1012.599,141.237,369.726,-28.588,52.388,-30.588
C06247=1012.597,141.501,369.699,-28.588,52.398,-30.584
C06248=1012.597,141.702,369.679,-28.588,52.407,-30.583
C06249=1012.596,142.102,369.638,-28.589,52.423,-30.578
C06250=1012.593,142.504,369.598,-28.590,52.440,-30.573
C06251=1012.592,142.905,369.557,-28.591,52.456,-30.570
C06252=1012.590,143.308,369.516,-28.592,52.472,-30.565
C06253=1012.588,143.711,369.475,-28.593,52.487,-30.562
C06254=1012.586,144.115,369.434,-28.593,52.504,-30.557
C06255=1012.585,144.519,369.393,-28.594,52.521,-30.553
C06256=1012.583,144.924,369.351,-28.595,52.538,-30.549
C06257=1012.581,145.330,369.310,-28.596,52.553,-30.545
C06258=1012.580,145.735,369.268,-28.597,52.570,-30.540
C06259=1012.578,146.141,369.227,-28.598,52.587,-30.536
C06260=1012.577,146.547,369.185,-28.598,52.603,-30.531
C06261=1012.575,146.955,369.144,-28.600,52.619,-30.528
C06262=1012.886,146.914,368.739,-27.647,41.032,-33.064
C06263=1012.888,146.506,368.780,-27.645,41.015,-33.069
C06264=1012.890,146.100,368.821,-27.643,40.999,-33.077
C06265=1012.891,145.694,368.863,-27.642,40.981,-33.084
C06266=1012.893,145.288,368.904,-27.640,40.965,-33.091
C06267=1012.895,144.883,368.946,-27.639,40.947,-33.098
C06268=1012.897,144.478,368.988,-27.637,40.932,-33.104
C06269=1012.898,144.074,369.028,-27.635,40.914,-33.111
C06270=1012.900,143.670,369.070,-27.634,40.898,-33.118
C06271=1012.902,143.267,369.111,-27.632,40.881,-33.125
C06272=1012.904,142.865,369.151,-27.631,40.864,-33.131
C06273=1012.906,142.463,369.193,-27.629,40.848,-33.139
C06274=1012.907,142.061,369.233,-27.627,40.832,-33.145
C06275=1012.909,141.661,369.274,-27.626,40.815,-33.153
C06276=1012.910,141.461,369.295,-27.625,40.807,-33.156
C06277=1012.911,141.196,369.322,-27.624,40.796,-33.161
C06278=1012.913,140.791,369.363,-27.623,40.780,-33.167
C06279=1012.914,140.573,369.385,-27.622,40.770,-33.171
C06280=1012.915,140.362,369.406,-27.621,40.762,-33.175
C06281=1012.915,140.135,369.429,-27.620,40.754,-33.178
C06282=1012.917,139.894,369.454,-27.619,40.743,-33.183
C06283=1012.918,139.639,369.480,-27.618,40.733,-33.187
C06284=1012.920,139.378,369.506,-27.617,40.723,-33.192
C06285=1012.920,139.117,369.533,-27.616,40.712,-33.196
C06286=1012.921,138.858,369.559,-27.615,40.702,-33.201
C06287=1012.923,138.610,369.584,-27.614,40.692,-33.205
C06288=1012.924,138.374,369.609,-27.613,40.682,-33.209
C06289=1012.925,138.155,369.631,-27.612,40.673,-33.212
C06290=1012.926,137.759,369.671,-27.611,40.657,-33.218
C06291=1012.928,137.458,369.701,-27.610,40.645,-33.224
C06292=1012.930,137.110,369.736,-27.608,40.632,-33.230
C06293=1012.931,136.767,369.771,-27.607,40.618,-33.235
C06294=1012.933,136.447,369.804,-27.606,40.604,-33.242
C06295=1012.934,136.125,369.837,-27.605,40.593,-33.247
C06296=1012.936,135.785,369.871,-27.603,40.578,-33.253
C06297=1012.937,135.416,369.908,-27.602,40.563,-33.260
C06298=1012.939,135.006,369.949,-27.600,40.546,-33.267
C06299=1012.940,134.746,369.976,-27.599,40.535,-33.271
C06300=1012.942,134.517,369.999,-27.598,40.525,-33.276
C06301=1012.943,134.121,370.039,-27.597,40.510,-33.283
C06302=1012.945,133.727,370.079,-27.595,40.494,-33.289
C06303=1012.947,133.333,370.118,-27.594,40.479,-33.295
C06304=1012.948,132.938,370.158,-27.592,40.465,-33.302
C06305=1012.950,132.544,370.198,-27.591,40.451,-33.308
C06306=1012.952,132.150,370.238,-27.589,40.434,-33.316
C06307=1012.953,131.756,370.277,-27.588,40.418,-33.322
C06308=1012.956,131.361,370.317,-27.586,40.402,-33.330
C06309=1012.957,130.967,370.357,-27.585,40.386,-33.337
C06310=1012.960,130.573,370.396,-27.583,40.370,-33.343
C06311=1012.961,130.179,370.436,-27.582,40.357,-33.350
C06312=1012.963,129.785,370.475,-27.580,40.342,-33.357
C06313=1012.964,129.390,370.516,-27.579,40.329,-33.363
C06314=1012.966,128.995,370.555,-27.577,40.314,-33.370
C06315=1012.967,128.602,370.595,-27.576,40.298,-33.376
C06316=1012.970,128.207,370.634,-27.574,40.281,-33.384
C06317=1012.971,127.813,370.673,-27.573,40.265,-33.391
C06318=1012.973,127.419,370.713,-27.571,40.250,-33.398
C06319=1012.975,127.024,370.753,-27.570,40.236,-33.404
C06320=1012.976,126.631,370.793,-27.568,40.221,-33.411
C06321=1012.978,126.236,370.832,-27.567,40.208,-33.417
C06322=1012.980,125.842,370.871,-27.566,40.195,-33.423
C06323=1012.982,125.448,370.911,-27.564,40.178,-33.431
C06324=1012.984,125.054,370.950,-27.562,40.162,-33.438
C06325=1012.985,124.659,370.989,-27.561,40.147,-33.445
C06326=1012.987,124.266,371.029,-27.559,40.132,-33.452
C06327=1012.989,123.872,371.068,-27.558,40.118,-33.457
C06328=1012.991,123.477,371.108,-27.557,40.103,-33.465
C06329=1012.993,123.084,371.147,-27.555,40.090,-33.471
C06330=1012.994,122.689,371.187,-27.554,40.077,-33.478
C06331=1012.996,122.295,371.226,-27.552,40.061,-33.485
C06332=1012.997,121.901,371.265,-27.551,40.046,-33.491
C06333=1012.999,121.507,371.305,-27.549,40.030,-33.498
C06334=1013.001,121.112,371.344,-27.548,40.015,-33.505
C06335=1013.003,120.718,371.383,-27.546,40.001,-33.513
C06336=1013.005,120.324,371.423,-27.545,39.988,-33.519
C06337=1013.007,119.930,371.462,-27.544,39.974,-33.525
C06338=1013.009,119.536,371.501,-27.542,39.961,-33.531
C06339=1013.010,119.142,371.540,-27.541,39.947,-33.539
C06340=1013.012,118.748,371.580,-27.539,39.931,-33.546
C06341=1013.013,118.354,371.619,-27.538,39.916,-33.553
C06342=1013.015,117.959,371.658,-27.536,39.902,-33.560
C06343=1013.017,117.566,371.697,-27.535,39.887,-33.566
C06344=1013.019,117.171,371.736,-27.534,39.873,-33.574
C06345=1013.021,116.777,371.775,-27.532,39.860,-33.580
C06346=1013.022,116.383,371.815,-27.531,39.847,-33.587
C06347=1013.024,115.989,371.854,-27.530,39.834,-33.593
C06348=1013.025,115.595,371.893,-27.528,39.819,-33.600
C06349=1013.028,115.201,371.932,-27.527,39.804,-33.607
C06350=1013.029,114.807,371.971,-27.525,39.789,-33.614
C06351=1013.031,114.412,372.010,-27.524,39.775,-33.620
C06352=1013.033,114.018,372.049,-27.522,39.761,-33.628
C06353=1013.034,113.624,372.088,-27.521,39.748,-33.634
C06354=1013.036,113.230,372.126,-27.520,39.736,-33.640
C06355=1013.038,112.836,372.165,-27.518,39.723,-33.647
C06356=1013.039,112.442,372.204,-27.517,39.708,-33.654
C06357=1013.041,112.047,372.243,-27.515,39.693,-33.661
C06358=1013.043,111.654,372.282,-27.514,39.679,-33.668
C06359=1013.045,111.259,372.321,-27.513,39.666,-33.675
C06360=1013.047,110.865,372.360,-27.511,39.652,-33.682
C06361=1013.048,110.471,372.399,-27.510,39.638,-33.689
C06362=1013.049,110.077,372.438,-27.509,39.626,-33.694
C06363=1013.051,109.683,372.476,-27.507,39.614,-33.701
C06364=1013.053,109.289,372.515,-27.506,39.600,-33.709
C06365=1013.055,108.894,372.555,-27.504,39.585,-33.716
C06366=1013.056,108.500,372.593,-27.503,39.571,-33.722
C06367=1013.058,108.107,372.632,-27.501,39.557,-33.730
C06368=1013.060,107.712,372.671,-27.500,39.544,-33.736
C06369=1013.061,107.318,372.710,-27.499,39.531,-33.743
C06370=1013.062,106.924,372.748,-27.497,39.519,-33.750
C06371=1013.064,106.529,372.787,-27.496,39.507,-33.755
C06372=1013.067,106.135,372.825,-27.495,39.494,-33.761
C06373=1013.068,105.741,372.865,-27.493,39.479,-33.769
C06374=1013.069,105.347,372.903,-27.492,39.465,-33.777
C06375=1013.071,104.953,372.942,-27.491,39.452,-33.783
C06376=1013.073,104.558,372.980,-27.489,39.438,-33.791
C06377=1013.074,104.164,373.019,-27.488,39.426,-33.796
C06378=1013.076,103.770,373.058,-27.487,39.413,-33.803
C06379=1013.078,103.376,373.097,-27.485,39.401,-33.810
C06380=1013.080,102.982,373.134,-27.484,39.390,-33.816
C06381=1013.081,102.587,373.173,-27.483,39.375,-33.823
C06382=1013.083,102.193,373.212,-27.481,39.361,-33.831
C06383=1013.084,101.798,373.250,-27.480,39.348,-33.837
C06384=1013.087,101.405,373.289,-27.478,39.335,-33.844
C06385=1013.088,101.010,373.328,-27.477,39.323,-33.851
C06386=1013.089,100.616,373.366,-27.476,39.310,-33.858
C06387=1013.091,100.221,373.405,-27.475,39.298,-33.863
C06388=1013.092,99.827,373.443,-27.473,39.287,-33.871
C06389=1013.095,99.433,373.481,-27.472,39.273,-33.877
C06390=1013.096,99.039,373.520,-27.470,39.259,-33.885
C06391=1013.098,98.644,373.558,-27.469,39.246,-33.891
C06392=1013.099,98.250,373.597,-27.468,39.233,-33.898
C06393=1013.100,97.855,373.635,-27.466,39.221,-33.905
C06394=1013.103,97.461,373.674,-27.465,39.208,-33.912
C06395=1013.104,97.067,373.712,-27.464,39.197,-33.918
C06396=1013.106,96.672,373.751,-27.463,39.186,-33.925
C06397=1013.107,96.276,373.789,-27.461,39.174,-33.931
C06398=1013.109,95.883,373.827,-27.460,39.160,-33.939
C06399=1013.110,95.490,373.865,-27.459,39.146,-33.945
C06400=1013.112,95.095,373.903,-27.457,39.133,-33.953
C06401=1013.113,94.701,373.942,-27.456,39.121,-33.959
C06402=1013.115,94.306,373.980,-27.455,39.109,-33.966
C06403=1013.117,93.911,374.018,-27.453,39.097,-33.973
C06404=1013.118,93.517,374.057,-27.452,39.086,-33.979
C06405=1013.120,93.122,374.095,-27.451,39.076,-33.985
C06406=1013.121,92.728,374.132,-27.450,39.063,-33.992
C06407=1013.123,92.334,374.171,-27.449,39.052,-33.998
C06408=1013.124,91.939,374.209,-27.447,39.038,-34.006
C06409=1013.126,91.544,374.247,-27.446,39.026,-34.013
C06410=1013.128,91.149,374.285,-27.444,39.013,-34.020
C06411=1013.129,90.747,374.325,-27.443,39.002,-34.027
C06412=1013.130,90.501,374.348,-27.442,38.994,-34.032
C06413=1013.131,90.222,374.375,-27.441,38.986,-34.036
C06414=1013.133,89.946,374.402,-27.441,38.979,-34.039
C06415=1013.133,89.712,374.425,-27.440,38.971,-34.043
C06416=1013.134,89.317,374.462,-27.439,38.961,-34.050
C06417=1013.136,88.932,374.499,-27.438,38.949,-34.057
C06418=1013.138,88.554,374.535,-27.436,38.938,-34.063
C06419=1013.139,88.179,374.572,-27.435,38.926,-34.070
C06420=1013.141,87.801,374.608,-27.434,38.915,-34.076
C06421=1013.142,87.417,374.646,-27.433,38.904,-34.082
C06422=1013.144,87.023,374.683,-27.431,38.892,-34.090
C06423=1013.145,86.624,374.721,-27.430,38.880,-34.097
C06424=1013.147,86.223,374.760,-27.429,38.869,-34.103
C06425=1013.148,85.822,374.799,-27.428,38.857,-34.110
C06426=1013.150,85.419,374.837,-27.426,38.845,-34.117
C06427=1013.151,85.015,374.876,-27.425,38.832,-34.124
C06428=1013.152,84.609,374.915,-27.424,38.822,-34.130
C06429=1013.154,84.202,374.954,-27.423,38.810,-34.138
C06430=1013.156,83.793,374.993,-27.421,38.798,-34.145
C06431=1013.157,83.384,375.032,-27.420,38.786,-34.152
C06432=1013.159,82.973,375.071,-27.419,38.773,-34.159
C06433=1013.160,82.561,375.111,-27.417,38.763,-34.165
C06434=1013.162,82.148,375.150,-27.416,38.751,-34.173
C06435=1013.164,81.735,375.190,-27.415,38.738,-34.180
C06436=1013.165,81.320,375.230,-27.414,38.727,-34.187
C06437=1013.167,80.926,375.267,-27.412,38.716,-34.193
C06438=1013.168,80.563,375.302,-27.411,38.705,-34.199
C06439=1013.169,80.180,375.339,-27.410,38.695,-34.206
C06440=1013.171,79.769,375.377,-27.409,38.683,-34.213
C06441=1013.172,79.359,375.417,-27.407,38.671,-34.220
C06442=1013.174,78.957,375.455,-27.406,38.660,-34.227
C06443=1013.175,78.562,375.493,-27.405,38.649,-34.234
C06444=1013.177,78.174,375.529,-27.404,38.639,-34.241
C06445=1013.178,77.790,375.566,-27.403,38.628,-34.247
C06446=1013.179,77.409,375.603,-27.401,38.617,-34.253
C06447=1013.181,77.027,375.639,-27.400,38.607,-34.260
C06448=1013.182,76.640,375.676,-27.399,38.596,-34.266
C06449=1013.183,76.247,375.713,-27.398,38.585,-34.273
C06450=1013.185,75.845,375.751,-27.397,38.575,-34.280
C06451=1013.186,75.436,375.790,-27.396,38.563,-34.287
C06452=1013.188,75.022,375.829,-27.394,38.552,-34.294
C06453=1013.189,74.813,375.848,-27.394,38.547,-34.297
C06454=1013.189,74.597,375.869,-27.393,38.541,-34.301
C06455=1013.190,74.371,375.890,-27.392,38.535,-34.305
C06456=1013.191,74.143,375.912,-27.392,38.528,-34.308
C06457=1013.191,73.924,375.933,-27.391,38.522,-34.312
C06458=1013.193,73.509,375.973,-27.390,38.511,-34.319
C06459=1013.195,73.098,376.011,-27.389,38.500,-34.327
C06460=1013.196,72.688,376.049,-27.387,38.489,-34.334
C06461=1013.198,72.281,376.089,-27.386,38.478,-34.340
C06462=1013.198,71.874,376.127,-27.385,38.468,-34.348
C06463=1013.200,71.470,376.165,-27.384,38.457,-34.354
C06464=1013.201,71.065,376.203,-27.382,38.445,-34.361
C06465=1013.203,70.660,376.242,-27.381,38.435,-34.368
C06466=1013.204,70.256,376.279,-27.380,38.425,-34.375
C06467=1013.206,69.852,376.317,-27.379,38.415,-34.381
C06468=1013.207,69.448,376.356,-27.378,38.404,-34.389
C06469=1013.208,69.040,376.394,-27.377,38.393,-34.395
C06470=1013.210,68.624,376.433,-27.375,38.383,-34.402
C06471=1013.211,68.206,376.473,-27.374,38.371,-34.409
C06472=1013.212,67.795,376.511,-27.373,38.362,-34.416
C06473=1013.214,67.394,376.549,-27.372,38.351,-34.422
C06474=1013.215,66.995,376.586,-27.371,38.340,-34.430
C06475=1013.216,66.599,376.623,-27.369,38.330,-34.437
C06476=1013.217,66.235,376.657,-27.368,38.321,-34.442
C06477=1013.219,65.908,376.689,-27.368,38.313,-34.448
C06478=1013.220,65.515,376.725,-27.366,38.303,-34.455
C06479=1013.220,65.307,376.744,-27.366,38.298,-34.457
C06480=1013.222,65.092,376.765,-27.365,38.293,-34.462
C06481=1013.222,64.873,376.786,-27.365,38.287,-34.465
C06482=1013.223,64.651,376.807,-27.364,38.281,-34.469
C06483=1013.223,64.425,376.827,-27.363,38.275,-34.473
C06484=1013.224,64.198,376.849,-27.363,38.270,-34.477
C06485=1013.225,63.979,376.870,-27.362,38.265,-34.481
C06486=1013.227,63.574,376.906,-27.355,38.206,-34.503
C06487=1013.231,63.363,376.922,-27.343,38.107,-34.538
C06488=1013.235,63.128,376.941,-27.330,37.997,-34.576
C06489=1013.239,62.880,376.961,-27.316,37.881,-34.616
C06490=1013.244,62.637,376.980,-27.302,37.769,-34.656
C06491=1013.247,62.418,376.997,-27.290,37.667,-34.691
C06492=1013.252,62.134,377.020,-27.273,37.536,-34.738
C06493=1013.258,61.736,377.052,-27.250,37.352,-34.805
C06494=1013.265,61.341,377.083,-27.227,37.169,-34.870
C06495=1013.272,60.944,377.115,-27.204,36.986,-34.936
C06496=1013.278,60.549,377.146,-27.181,36.805,-35.002
C06497=1013.285,60.153,377.178,-27.157,36.624,-35.068
C06498=1013.291,59.757,377.210,-27.134,36.443,-35.134
C06499=1013.298,59.361,377.241,-27.110,36.263,-35.201
C06500=1013.304,58.965,377.273,-27.086,36.082,-35.268
C06501=1013.312,58.569,377.305,-27.062,35.903,-35.336
C06502=1013.317,58.173,377.336,-27.038,35.724,-35.405
C06503=1013.324,57.778,377.368,-27.014,35.546,-35.472
C06504=1013.331,57.382,377.400,-26.989,35.368,-35.541
C06505=1013.337,56.986,377.431,-26.965,35.191,-35.609
C06506=1013.344,56.591,377.463,-26.940,35.013,-35.680
C06507=1013.350,56.194,377.495,-26.915,34.837,-35.749
C06508=1013.357,55.799,377.526,-26.890,34.661,-35.818
C06509=1013.363,55.402,377.558,-26.865,34.485,-35.888
C06510=1013.370,55.007,377.590,-26.839,34.311,-35.959
C06511=1013.376,54.611,377.621,-26.814,34.137,-36.028
C06512=1013.383,54.215,377.653,-26.788,33.962,-36.099
C06513=1013.389,53.819,377.686,-26.763,33.790,-36.170
C06514=1013.396,53.423,377.717,-26.737,33.617,-36.240
C06515=1013.402,53.028,377.749,-26.711,33.445,-36.312
C06516=1013.409,52.632,377.781,-26.684,33.274,-36.383
C06517=1013.415,52.237,377.812,-26.658,33.103,-36.454
C06518=1013.422,51.840,377.844,-26.632,32.933,-36.527
C06519=1013.428,51.445,377.875,-26.605,32.763,-36.598
C06520=1013.434,51.049,377.908,-26.578,32.594,-36.670
C06521=1013.441,50.653,377.939,-26.552,32.426,-36.743
C06522=1013.447,50.258,377.971,-26.525,32.258,-36.816
C06523=1013.454,49.862,378.004,-26.498,32.091,-36.888
C06524=1013.460,49.466,378.035,-26.470,31.925,-36.961
C06525=1013.466,49.071,378.067,-26.443,31.758,-37.035
C06526=1013.472,48.675,378.098,-26.415,31.593,-37.108
C06527=1013.479,48.280,378.131,-26.388,31.430,-37.181
C06528=1013.485,47.884,378.163,-26.360,31.265,-37.255
C06529=1013.492,47.488,378.194,-26.332,31.102,-37.330
C06530=1013.498,47.092,378.227,-26.304,30.939,-37.403
C06531=1013.504,46.698,378.258,-26.276,30.776,-37.477
C06532=1013.510,46.301,378.290,-26.248,30.615,-37.552
C06533=1013.517,45.906,378.322,-26.220,30.454,-37.627
C06534=1013.522,45.511,378.354,-26.191,30.294,-37.701
C06535=1013.529,45.115,378.386,-26.163,30.135,-37.776
C06536=1013.535,44.719,378.418,-26.134,29.976,-37.852
C06537=1013.542,44.324,378.450,-26.105,29.818,-37.926
C06538=1013.547,43.929,378.482,-26.076,29.659,-38.001
C06539=1013.554,43.533,378.514,-26.047,29.502,-38.078
C06540=1013.559,43.138,378.546,-26.018,29.346,-38.153
C06541=1013.565,42.743,378.578,-25.989,29.190,-38.228
C06542=1013.572,42.346,378.610,-25.959,29.035,-38.305
C06543=1013.578,41.952,378.641,-25.930,28.881,-38.381
C06544=1013.584,41.556,378.673,-25.900,28.726,-38.458
C06545=1013.590,41.161,378.705,-25.871,28.573,-38.534
C06546=1013.596,40.765,378.737,-25.841,28.421,-38.610
C06547=1013.602,40.370,378.769,-25.811,28.269,-38.686
C06548=1013.608,39.974,378.802,-25.781,28.117,-38.763
C06549=1013.614,39.580,378.833,-25.751,27.967,-38.840
C06550=1013.620,39.184,378.865,-25.721,27.817,-38.916
C06551=1013.626,38.789,378.897,-25.690,27.667,-38.994
C06552=1013.632,38.393,378.930,-25.660,27.519,-39.070
C06553=1013.638,37.998,378.961,-25.629,27.371,-39.148
C06554=1013.643,37.603,378.994,-25.599,27.224,-39.224
C06555=1013.649,37.209,379.026,-25.568,27.077,-39.303
C06556=1013.655,36.813,379.058,-25.537,26.931,-39.381
C06557=1013.662,36.418,379.090,-25.506,26.785,-39.457
C06558=1013.667,36.022,379.122,-25.475,26.640,-39.535
C06559=1013.673,35.627,379.154,-25.444,26.496,-39.612
C06560=1013.679,35.232,379.186,-25.413,26.353,-39.690
C06561=1013.684,34.837,379.218,-25.382,26.211,-39.768
C06562=1013.690,34.442,379.250,-25.350,26.069,-39.847
C06563=1013.696,34.046,379.282,-25.319,25.927,-39.924
C06564=1013.702,33.652,379.314,-25.287,25.786,-40.003
C06565=1013.707,33.257,379.346,-25.256,25.647,-40.080
C06566=1013.712,32.861,379.378,-25.224,25.507,-40.158
C06567=1013.718,32.466,379.410,-25.192,25.368,-40.237
C06568=1013.724,32.071,379.443,-25.160,25.230,-40.315
C06569=1013.729,31.676,379.475,-25.129,25.093,-40.393
C06570=1013.735,31.281,379.506,-25.097,24.956,-40.472
C06571=1013.740,30.886,379.539,-25.065,24.820,-40.549
C06572=1013.746,30.491,379.571,-25.033,24.685,-40.628
C06573=1013.752,30.095,379.603,-25.001,24.551,-40.706
C06574=1013.757,29.701,379.636,-24.968,24.416,-40.784
C06575=1013.763,29.306,379.667,-24.936,24.283,-40.863
C06576=1013.769,28.910,379.699,-24.904,24.151,-40.942
C06577=1013.773,28.515,379.731,-24.871,24.019,-41.020
C06578=1013.780,28.122,379.763,-24.839,23.888,-41.097
C06579=1013.785,27.729,379.795,-24.807,23.759,-41.176
C06580=1013.789,27.337,379.827,-24.774,23.630,-41.254
C06581=1013.795,26.943,379.859,-24.742,23.501,-41.332
C06582=1013.800,26.549,379.891,-24.709,23.373,-41.410
C06583=1013.806,26.153,379.923,-24.677,23.245,-41.489
C06584=1013.811,25.755,379.956,-24.644,23.117,-41.568
C06585=1013.816,25.357,379.988,-24.611,22.990,-41.647
C06586=1013.821,24.961,380.021,-24.578,22.864,-41.725
C06587=1013.827,24.566,380.053,-24.545,22.739,-41.803
C06588=1013.832,24.170,380.084,-24.512,22.615,-41.881
C06589=1013.837,23.792,380.115,-24.481,22.496,-41.956
C06590=1013.841,23.451,380.143,-24.452,22.390,-42.024
C06591=1013.847,23.036,380.177,-24.418,22.262,-42.106
C06592=1013.851,22.672,380.206,-24.387,22.150,-42.178
C06593=1013.855,22.395,380.230,-24.364,22.065,-42.232
C06594=1013.858,22.064,380.256,-24.337,21.965,-42.297
C06595=1013.863,21.737,380.283,-24.309,21.865,-42.363
C06596=1013.868,21.348,380.314,-24.277,21.748,-42.438
C06597=1013.871,21.121,380.333,-24.258,21.680,-42.483
C06598=1013.876,20.700,380.367,-24.222,21.554,-42.566
C06599=1013.879,20.523,380.381,-24.208,21.502,-42.601
C06600=1013.892,19.425,380.471,-24.206,21.503,-42.613
C06601=1013.897,19.077,380.499,-24.205,21.502,-42.619
C06602=1013.900,18.745,380.525,-24.205,21.503,-42.622
C06603=1013.904,18.413,380.552,-24.204,21.503,-42.626
C06604=1013.909,18.082,380.579,-24.204,21.504,-42.630
C06605=1013.912,17.751,380.606,-24.203,21.504,-42.634
C06606=1013.916,17.421,380.634,-24.202,21.504,-42.639
C06607=1013.920,17.091,380.660,-24.202,21.505,-42.643
C06608=1013.924,16.762,380.687,-24.201,21.505,-42.646
C06609=1013.927,16.434,380.714,-24.201,21.506,-42.650
C06610=1013.931,16.106,380.740,-24.200,21.506,-42.654
C06611=1013.935,15.778,380.766,-24.200,21.507,-42.658
C06612=1013.939,15.452,380.793,-24.199,21.507,-42.663
C06613=1013.943,15.125,380.820,-24.199,21.507,-42.667
C06614=1013.946,14.799,380.847,-24.198,21.508,-42.670
C06615=1013.950,14.474,380.873,-24.198,21.508,-42.674
C06616=1013.954,14.149,380.899,-24.197,21.509,-42.678
C06617=1013.957,13.824,380.925,-24.197,21.509,-42.682
C06618=1013.961,13.500,380.951,-24.196,21.509,-42.687
C06619=1013.964,13.176,380.978,-24.195,21.509,-42.691
C06620=1013.968,12.852,381.003,-24.195,21.510,-42.694
C06621=1013.972,12.529,381.030,-24.194,21.510,-42.698
C06622=1013.975,12.205,381.057,-24.194,21.511,-42.702
C06623=1013.978,11.881,381.082,-24.193,21.511,-42.707
C06624=1013.982,11.559,381.108,-24.193,21.511,-42.711
C06625=1013.985,11.235,381.135,-24.192,21.512,-42.715
C06626=1013.988,10.913,381.161,-24.192,21.512,-42.718
C06627=1013.991,10.592,381.187,-24.191,21.513,-42.722
C06628=1013.995,10.273,381.213,-24.191,21.513,-42.726
C06629=1013.998,9.957,381.238,-24.190,21.514,-42.730
C06630=1014.002,9.641,381.264,-24.190,21.514,-42.733
C06631=1014.005,9.327,381.290,-24.189,21.514,-42.738
C06632=1014.007,9.012,381.315,-24.188,21.515,-42.742
C06633=1014.011,8.697,381.340,-24.188,21.515,-42.746
C06634=1014.014,8.381,381.366,-24.187,21.516,-42.750
C06635=1014.017,8.063,381.392,-24.186,21.515,-42.755
C06636=1014.020,7.742,381.418,-24.186,21.516,-42.759
C06637=1014.023,7.418,381.444,-24.186,21.516,-42.762
C06638=1014.026,7.093,381.470,-24.185,21.517,-42.766
C06639=1014.030,6.766,381.497,-24.185,21.517,-42.770
C06640=1014.033,6.438,381.522,-24.184,21.518,-42.774
C06641=1014.036,6.109,381.549,-24.183,21.518,-42.779
C06642=1014.039,5.779,381.576,-24.183,21.518,-42.783
C06643=1014.042,5.450,381.603,-24.182,21.519,-42.786
C06644=1014.045,5.120,381.630,-24.181,21.518,-42.792
C06645=1014.048,4.788,381.656,-24.181,21.519,-42.795
C06646=1014.051,4.458,381.683,-24.180,21.519,-42.799
C06647=1014.054,4.126,381.709,-24.180,21.521,-42.803
C06648=1014.057,3.796,381.736,-24.179,21.520,-42.807
C06649=1014.060,3.484,381.761,-24.179,21.521,-42.810
C06650=1014.062,3.194,381.784,-24.179,21.521,-42.814
C06651=1014.065,2.924,381.807,-24.178,21.522,-42.818
C06652=1014.067,2.663,381.827,-24.177,21.522,-42.823
C06653=1014.069,2.394,381.849,-24.177,21.522,-42.827
C06654=1014.072,2.106,381.872,-24.176,21.523,-42.831
C06655=1014.074,1.793,381.897,-24.176,21.523,-42.834
C06656=1014.077,1.463,381.923,-24.175,21.523,-42.838
C06657=1014.080,1.129,381.951,-24.175,21.524,-42.842
C06658=1014.082,0.796,381.977,-24.174,21.525,-42.846
C06659=1014.085,0.461,382.005,-24.173,21.525,-42.851
C06660=1014.089,0.125,382.031,-24.173,21.525,-42.855
C06661=1014.091,-0.212,382.059,-24.172,21.526,-42.858
C06662=1014.094,-0.550,382.086,-24.172,21.526,-42.864
C06663=1014.096,-0.890,382.113,-24.171,21.526,-42.867
C06664=1014.100,-1.232,382.141,-24.170,21.527,-42.873
C06665=1014.101,-1.575,382.168,-24.170,21.527,-42.877
C06666=1014.105,-1.921,382.196,-24.169,21.528,-42.880
C06667=1014.107,-2.267,382.224,-24.169,21.528,-42.886
C06668=1014.109,-2.615,382.252,-24.168,21.529,-42.890
C06669=1014.113,-2.965,382.279,-24.167,21.529,-42.895
C06670=1014.115,-3.316,382.308,-24.167,21.529,-42.899
C06671=1014.117,-3.669,382.337,-24.166,21.529,-42.904
C06672=1014.120,-4.023,382.365,-24.166,21.531,-42.908
C06673=1014.123,-4.381,382.393,-24.165,21.530,-42.913
C06674=1014.126,-4.742,382.422,-24.164,21.531,-42.919
C06675=1014.128,-5.108,382.452,-24.164,21.532,-42.923
C06676=1014.131,-5.478,382.481,-24.163,21.532,-42.928
C06677=1014.134,-5.852,382.511,-24.163,21.533,-42.932
C06678=1014.136,-6.227,382.541,-24.162,21.533,-42.937
C06679=1014.139,-6.603,382.571,-24.161,21.533,-42.941
C06680=1014.142,-6.977,382.601,-24.160,21.534,-42.947
C06681=1014.144,-7.349,382.631,-24.160,21.534,-42.952
C06682=1014.146,-7.718,382.660,-24.159,21.535,-42.956
C06683=1014.149,-8.083,382.690,-24.158,21.535,-42.961
C06684=1014.151,-8.447,382.719,-24.158,21.536,-42.967
C06685=1014.153,-8.810,382.748,-24.157,21.536,-42.971
C06686=1014.156,-9.173,382.776,-24.156,21.536,-42.976
C06687=1014.158,-9.535,382.805,-24.156,21.537,-42.982
C06688=1014.160,-9.897,382.834,-24.155,21.538,-42.985
C06689=1014.162,-10.259,382.863,-24.154,21.538,-42.991
C06690=1014.165,-10.620,382.892,-24.154,21.539,-42.995
C06691=1014.167,-10.979,382.920,-24.153,21.539,-43.000
C06692=1014.169,-11.338,382.949,-24.152,21.539,-43.006
C06693=1014.171,-11.697,382.978,-24.152,21.540,-43.009
C06694=1014.174,-12.052,383.006,-24.151,21.540,-43.014
C06695=1014.175,-12.407,383.034,-24.151,21.541,-43.019
C06696=1014.177,-12.761,383.063,-24.150,21.541,-43.024
C06697=1014.179,-13.112,383.091,-24.149,21.542,-43.028
C06698=1014.181,-13.463,383.119,-24.149,21.542,-43.033
C06699=1014.183,-13.811,383.147,-24.148,21.543,-43.037
C06700=1014.185,-14.157,383.174,-24.147,21.543,-43.042
C06701=1014.187,-14.501,383.201,-24.147,21.544,-43.046
C06702=1014.188,-14.843,383.228,-24.146,21.544,-43.052
C06703=1014.190,-15.184,383.255,-24.146,21.544,-43.055
C06704=1014.192,-15.521,383.282,-24.145,21.545,-43.061
C06705=1014.193,-15.858,383.308,-24.145,21.546,-43.065
C06706=1014.195,-16.193,383.335,-24.144,21.546,-43.070
C06707=1014.197,-16.528,383.362,-24.143,21.546,-43.074
C06708=1014.199,-16.861,383.388,-24.142,21.547,-43.079
C06709=1014.200,-17.194,383.415,-24.142,21.547,-43.083
C06710=1014.202,-17.527,383.441,-24.141,21.547,-43.088
C06711=1014.204,-17.860,383.467,-24.141,21.548,-43.092
C06712=1014.205,-18.225,383.497,-24.140,21.549,-43.100
C06713=1014.206,-18.447,383.514,-24.139,21.548,-43.103
C06714=1014.207,-18.695,383.534,-24.139,21.549,-43.105
C06715=1014.209,-18.956,383.555,-24.139,21.550,-43.107
C06716=1014.209,-19.217,383.575,-24.139,21.550,-43.109
C06717=1014.211,-19.466,383.595,-24.138,21.550,-43.112
C06718=1014.213,-19.882,383.627,-24.137,21.550,-43.118
C06719=1014.214,-20.054,383.641,-24.137,21.551,-43.122
C06720=1014.215,-20.387,383.667,-24.136,21.551,-43.127
C06721=1014.216,-20.720,383.694,-24.136,21.552,-43.131
C06722=1014.218,-21.052,383.720,-24.135,21.553,-43.135
C06723=1014.219,-21.386,383.746,-24.134,21.552,-43.140
C06724=1014.220,-21.718,383.773,-24.134,21.553,-43.144
C06725=1014.222,-22.051,383.798,-24.133,21.554,-43.149
C06726=1014.223,-22.383,383.825,-24.133,21.554,-43.153
C06727=1014.224,-22.716,383.852,-24.132,21.554,-43.158
C06728=1014.225,-23.050,383.878,-24.131,21.556,-43.162
C06729=1014.227,-23.382,383.904,-24.131,21.555,-43.168
C06730=1014.228,-23.715,383.930,-24.130,21.556,-43.171
C06731=1014.229,-24.047,383.956,-24.129,21.556,-43.177
C06732=1014.230,-24.381,383.982,-24.129,21.557,-43.181
C06733=1014.231,-24.713,384.008,-24.128,21.557,-43.186
C06734=1014.233,-25.046,384.035,-24.128,21.558,-43.190
C06735=1014.233,-25.379,384.061,-24.127,21.558,-43.195
C06736=1014.235,-25.712,384.088,-24.126,21.559,-43.199
C06737=1014.236,-26.044,384.113,-24.126,21.559,-43.204
C06738=1014.237,-26.376,384.139,-24.125,21.559,-43.208
C06739=1014.238,-26.710,384.165,-24.124,21.560,-43.214
C06740=1014.239,-27.042,384.191,-24.124,21.560,-43.217
C06741=1014.240,-27.375,384.218,-24.123,21.560,-43.223
C06742=1014.241,-27.708,384.244,-24.123,21.562,-43.227
C06743=1014.242,-28.040,384.270,-24.122,21.562,-43.232
C06744=1014.243,-28.373,384.295,-24.121,21.562,-43.236
C06745=1014.244,-28.706,384.322,-24.120,21.562,-43.241
C06746=1014.244,-29.039,384.349,-24.120,21.563,-43.245
C06747=1014.245,-29.372,384.374,-24.119,21.563,-43.250
C06748=1014.246,-29.704,384.400,-24.119,21.564,-43.254
C06749=1014.247,-30.038,384.426,-24.118,21.565,-43.260
C06750=1014.248,-30.369,384.452,-24.118,21.565,-43.264
C06751=1014.249,-30.702,384.479,-24.117,21.565,-43.269
C06752=1014.250,-31.035,384.504,-24.116,21.566,-43.273
C06753=1014.250,-31.368,384.531,-24.116,21.566,-43.278
C06754=1014.251,-31.701,384.556,-24.115,21.567,-43.282
C06755=1014.252,-32.033,384.582,-24.114,21.567,-43.287
C06756=1014.252,-32.366,384.609,-24.114,21.568,-43.291
C06757=1014.253,-32.699,384.634,-24.113,21.568,-43.296
C06758=1014.253,-33.032,384.661,-24.113,21.569,-43.301
C06759=1014.254,-33.365,384.686,-24.112,21.569,-43.306
C06760=1014.255,-33.697,384.712,-24.111,21.570,-43.310
C06761=1014.254,-34.030,384.738,-24.111,21.570,-43.315
C06762=1014.255,-34.363,384.764,-24.110,21.571,-43.319
C06763=1014.256,-34.695,384.790,-24.109,21.571,-43.324
C06764=1014.256,-35.028,384.816,-24.109,21.572,-43.328
C06765=1014.257,-35.361,384.842,-24.108,21.572,-43.334
C06766=1014.258,-35.693,384.868,-24.108,21.573,-43.337
C06767=1014.258,-36.026,384.893,-24.107,21.573,-43.343
C06768=1014.258,-36.359,384.919,-24.107,21.574,-43.347
C06769=1014.259,-36.691,384.946,-24.106,21.574,-43.352
C06770=1014.259,-37.024,384.971,-24.105,21.574,-43.357
C06771=1014.259,-37.357,384.997,-24.105,21.575,-43.361
C06772=1014.260,-37.689,385.023,-24.104,21.575,-43.366
C06773=1014.260,-38.022,385.048,-24.103,21.576,-43.371
C06774=1014.260,-38.354,385.074,-24.102,21.576,-43.376
C06775=1014.261,-38.688,385.100,-24.102,21.577,-43.380
C06776=1014.261,-39.020,385.126,-24.101,21.577,-43.385
C06777=1014.262,-39.352,385.152,-24.101,21.578,-43.389
C06778=1014.262,-39.685,385.177,-24.100,21.578,-43.394
C06779=1014.262,-40.018,385.203,-24.100,21.579,-43.398
C06780=1014.262,-40.350,385.229,-24.099,21.579,-43.404
C06781=1014.263,-40.683,385.255,-24.098,21.580,-43.409
C06782=1014.262,-41.016,385.281,-24.098,21.580,-43.413
C06783=1014.262,-41.348,385.306,-24.097,21.580,-43.418
C06784=1014.262,-41.681,385.332,-24.096,21.582,-43.422
C06785=1014.262,-42.013,385.358,-24.096,21.582,-43.427
C06786=1014.262,-42.346,385.383,-24.095,21.582,-43.431
C06787=1014.263,-42.679,385.409,-24.094,21.583,-43.437
C06788=1014.263,-43.011,385.434,-24.094,21.583,-43.442
C06789=1014.262,-43.343,385.460,-24.093,21.583,-43.446
C06790=1014.263,-43.676,385.486,-24.092,21.584,-43.451
C06791=1014.262,-44.009,385.512,-24.092,21.585,-43.455
C06792=1014.262,-44.341,385.537,-24.091,21.585,-43.461
C06793=1014.262,-44.674,385.562,-24.091,21.586,-43.465
C06794=1014.262,-45.006,385.588,-24.090,21.586,-43.470
C06795=1014.262,-45.339,385.614,-24.089,21.586,-43.475
C06796=1014.262,-45.671,385.640,-24.089,21.587,-43.479
C06797=1014.262,-46.005,385.665,-24.088,21.588,-43.485
C06798=1014.261,-46.337,385.691,-24.088,21.588,-43.488
C06799=1014.261,-46.669,385.717,-24.087,21.588,-43.494
C06800=1014.261,-47.002,385.742,-24.086,21.590,-43.498
C06801=1014.261,-47.334,385.767,-24.086,21.589,-43.503
C06802=1014.260,-47.667,385.794,-24.085,21.589,-43.508
C06803=1014.260,-47.999,385.819,-24.084,21.591,-43.512
C06804=1014.259,-48.332,385.844,-24.083,21.591,-43.518
C06805=1014.259,-48.664,385.869,-24.083,21.592,-43.522
C06806=1014.259,-48.996,385.895,-24.082,21.592,-43.527
C06807=1014.258,-49.330,385.920,-24.081,21.592,-43.532
C06808=1014.258,-49.662,385.946,-24.081,21.593,-43.536
C06809=1014.258,-49.994,385.972,-24.080,21.593,-43.542
C06810=1014.257,-50.326,385.997,-24.080,21.595,-43.546
C06811=1014.257,-50.659,386.022,-24.079,21.594,-43.551
C06812=1014.256,-50.992,386.048,-24.079,21.595,-43.555
C06813=1014.256,-51.324,386.074,-24.078,21.596,-43.560
C06814=1014.255,-51.656,386.099,-24.077,21.596,-43.566
C06815=1014.255,-51.988,386.124,-24.077,21.597,-43.570
C06816=1014.254,-52.320,386.149,-24.076,21.597,-43.575
C06817=1014.253,-52.653,386.175,-24.075,21.597,-43.579
C06818=1014.253,-52.986,386.200,-24.075,21.598,-43.584
C06819=1014.252,-53.317,386.226,-24.074,21.598,-43.589
C06820=1014.252,-53.650,386.251,-24.074,21.600,-43.594
C06821=1014.251,-53.981,386.276,-24.073,21.599,-43.599
C06822=1014.250,-54.315,386.302,-24.072,21.600,-43.603
C06823=1014.249,-54.647,386.327,-24.072,21.601,-43.608
C06824=1014.248,-54.979,386.352,-24.071,21.601,-43.613
C06825=1014.248,-55.312,386.378,-24.070,21.602,-43.618
C06826=1014.247,-55.644,386.402,-24.070,21.602,-43.623
C06827=1014.246,-55.977,386.428,-24.069,21.603,-43.627
C06828=1014.245,-56.309,386.453,-24.068,21.603,-43.632
C06829=1014.245,-56.643,386.479,-24.068,21.603,-43.637
C06830=1014.244,-56.976,386.504,-24.067,21.605,-43.642
C06831=1014.243,-57.309,386.530,-24.066,21.604,-43.647
C06832=1014.241,-57.643,386.555,-24.066,21.605,-43.652
C06833=1014.241,-57.976,386.581,-24.065,21.606,-43.656
C06834=1014.240,-58.311,386.606,-24.064,21.606,-43.662
C06835=1014.239,-58.646,386.631,-24.064,21.607,-43.666
C06836=1014.238,-58.980,386.656,-24.063,21.607,-43.671
C06837=1014.237,-59.316,386.682,-24.062,21.608,-43.676
C06838=1014.235,-59.652,386.707,-24.062,21.608,-43.680
C06839=1014.235,-59.988,386.733,-24.061,21.609,-43.686
C06840=1014.233,-60.324,386.758,-24.060,21.609,-43.691
C06841=1014.233,-60.661,386.783,-24.060,21.610,-43.695
C06842=1014.231,-60.999,386.809,-24.059,21.610,-43.700
C06843=1014.230,-61.336,386.835,-24.059,21.611,-43.706
C06844=1014.229,-61.674,386.861,-24.058,21.611,-43.710
C06845=1014.227,-62.013,386.886,-24.057,21.612,-43.715
C06846=1014.226,-62.351,386.911,-24.057,21.612,-43.720
C06847=1014.225,-62.691,386.937,-24.056,21.614,-43.725
C06848=1014.223,-63.030,386.963,-24.055,21.613,-43.730
C06849=1014.222,-63.370,386.989,-24.055,21.614,-43.735
C06850=1014.221,-63.710,387.014,-24.054,21.615,-43.739
C06851=1014.219,-64.051,387.039,-24.053,21.616,-43.745
C06852=1014.218,-64.392,387.065,-24.053,21.615,-43.750
C06853=1014.216,-64.733,387.091,-24.052,21.617,-43.754
C06854=1014.214,-65.075,387.117,-24.051,21.617,-43.759
C06855=1014.213,-65.416,387.143,-24.051,21.618,-43.765
C06856=1014.212,-65.759,387.169,-24.050,21.617,-43.770
C06857=1014.211,-66.101,387.194,-24.050,21.619,-43.774
C06858=1014.208,-66.444,387.220,-24.049,21.619,-43.780
C06859=1014.207,-66.787,387.246,-24.048,21.620,-43.785
C06860=1014.205,-67.130,387.272,-24.048,21.620,-43.789
C06861=1014.205,-67.473,387.297,-24.047,21.621,-43.795
C06862=1014.202,-67.816,387.323,-24.046,21.621,-43.800
C06863=1014.201,-68.160,387.349,-24.045,21.622,-43.805
C06864=1014.199,-68.503,387.375,-24.045,21.622,-43.809
C06865=1014.197,-68.847,387.401,-24.044,21.623,-43.815
C06866=1014.195,-69.191,387.426,-24.043,21.623,-43.820
C06867=1014.194,-69.535,387.452,-24.043,21.624,-43.824
C06868=1014.192,-69.879,387.478,-24.042,21.624,-43.829
C06869=1014.189,-70.223,387.504,-24.041,21.625,-43.835
C06870=1014.188,-70.567,387.530,-24.041,21.625,-43.840
C06871=1014.186,-70.911,387.555,-24.040,21.626,-43.844
C06872=1014.184,-71.255,387.581,-24.040,21.627,-43.850
C06873=1014.182,-71.600,387.607,-24.039,21.627,-43.855
C06874=1014.181,-71.944,387.632,-24.038,21.628,-43.861
C06875=1014.178,-72.288,387.658,-24.038,21.628,-43.865
C06876=1014.176,-72.633,387.684,-24.037,21.629,-43.870
C06877=1014.174,-72.976,387.710,-24.036,21.629,-43.875
C06878=1014.172,-73.320,387.736,-24.035,21.630,-43.881
C06879=1014.170,-73.664,387.761,-24.035,21.630,-43.885
C06880=1014.168,-74.007,387.786,-24.034,21.631,-43.890
C06881=1014.165,-74.351,387.813,-24.033,21.632,-43.896
C06882=1014.164,-74.695,387.839,-24.033,21.632,-43.901
C06883=1014.162,-75.039,387.864,-24.032,21.633,-43.905
C06884=1014.159,-75.382,387.890,-24.031,21.633,-43.911
C06885=1014.157,-75.725,387.916,-24.031,21.634,-43.916
C06886=1014.154,-76.068,387.940,-24.030,21.634,-43.920
C06887=1014.152,-76.411,387.966,-24.030,21.635,-43.926
C06888=1014.150,-76.754,387.992,-24.029,21.635,-43.931
C06889=1014.147,-77.097,388.017,-24.028,21.636,-43.936
C06890=1014.145,-77.439,388.043,-24.028,21.636,-43.940
C06891=1014.142,-77.780,388.068,-24.027,21.637,-43.946
C06892=1014.140,-78.122,388.093,-24.026,21.637,-43.951
C06893=1014.138,-78.464,388.119,-24.026,21.639,-43.955
C06894=1014.135,-78.805,388.145,-24.025,21.638,-43.960
C06895=1014.132,-79.146,388.170,-24.024,21.639,-43.966
C06896=1014.130,-79.486,388.195,-24.023,21.639,-43.971
C06897=1014.128,-79.827,388.220,-24.023,21.641,-43.975
C06898=1014.125,-80.167,388.246,-24.022,21.641,-43.981
C06899=1014.122,-80.506,388.271,-24.021,21.641,-43.986
C06900=1014.119,-80.845,388.296,-24.021,21.643,-43.990
C06901=1014.117,-81.184,388.321,-24.020,21.643,-43.995
C06902=1014.114,-81.523,388.346,-24.020,21.643,-44.001
C06903=1014.112,-81.860,388.371,-24.019,21.644,-44.005
C06904=1014.109,-82.198,388.396,-24.018,21.645,-44.010
C06905=1014.106,-82.535,388.421,-24.018,21.645,-44.016
C06906=1014.103,-82.871,388.446,-24.017,21.645,-44.021
C06907=1014.101,-83.207,388.470,-24.016,21.646,-44.025
C06908=1014.098,-83.543,388.495,-24.016,21.647,-44.031
C06909=1014.095,-83.879,388.521,-24.015,21.647,-44.036
C06910=1014.092,-84.214,388.545,-24.015,21.648,-44.040
C06911=1014.090,-84.547,388.570,-24.014,21.648,-44.045
C06912=1014.086,-84.898,388.596,-24.013,21.649,-44.051
C06913=1014.083,-85.294,388.625,-24.012,21.650,-44.056
C06914=1014.081,-85.507,388.641,-24.012,21.649,-44.060
C06915=1014.079,-85.720,388.656,-24.012,21.649,-44.062
C06916=1014.076,-86.129,388.687,-24.011,21.650,-44.067
C06917=1014.072,-86.489,388.714,-24.010,21.651,-44.073
C06918=1014.070,-86.819,388.738,-24.009,21.652,-44.078
C06919=1014.067,-87.141,388.762,-24.009,21.652,-44.082
C06920=1014.063,-87.457,388.785,-24.008,21.653,-44.088
C06921=1014.060,-87.770,388.807,-24.007,21.653,-44.093
C06922=1014.057,-88.081,388.831,-24.007,21.654,-44.097
C06923=1014.054,-88.393,388.854,-24.006,21.654,-44.102
C06924=1014.051,-88.712,388.878,-24.006,21.655,-44.106
C06925=1014.048,-89.083,388.904,-24.005,21.656,-44.114
C06926=1014.046,-89.302,388.921,-24.004,21.656,-44.117
C06927=1014.043,-89.537,388.938,-24.004,21.656,-44.119
C06928=1014.041,-89.775,388.956,-24.004,21.656,-44.121
C06929=1014.038,-90.005,388.973,-24.004,21.657,-44.123
C06930=1014.034,-90.412,389.003,-24.003,21.658,-44.130
C06931=1014.031,-90.749,389.028,-24.002,21.658,-44.136
C06932=1014.027,-91.079,389.052,-24.001,21.659,-44.141
C06933=1014.024,-91.408,389.076,-24.001,21.660,-44.145
C06934=1014.021,-91.737,389.100,-24.000,21.660,-44.150
C06935=1014.017,-92.066,389.124,-23.999,21.660,-44.156
C06936=1014.014,-92.394,389.149,-23.999,21.661,-44.160
C06937=1014.011,-92.721,389.173,-23.998,21.662,-44.165
C06938=1014.007,-93.048,389.197,-23.998,21.662,-44.169
C06939=1014.003,-93.375,389.220,-23.997,21.663,-44.175
C06940=1014.000,-93.700,389.244,-23.996,21.663,-44.180
C06941=1013.996,-94.025,389.268,-23.996,21.664,-44.184
C06942=1013.992,-94.350,389.293,-23.995,21.664,-44.189
C06943=1013.990,-94.674,389.316,-23.994,21.665,-44.193
C06944=1013.986,-94.998,389.340,-23.994,21.666,-44.199
C06945=1013.982,-95.321,389.364,-23.993,21.666,-44.204
C06946=1013.978,-95.644,389.387,-23.993,21.666,-44.207
C06947=1013.975,-95.966,389.411,-23.992,21.667,-44.213
C06948=1013.970,-96.288,389.434,-23.991,21.668,-44.217
C06949=1013.967,-96.609,389.458,-23.991,21.668,-44.222
C06950=1013.964,-96.931,389.481,-23.990,21.669,-44.226
C06951=1013.960,-97.253,389.506,-23.989,21.669,-44.231
C06952=1013.956,-97.574,389.528,-23.989,21.670,-44.236
C06953=1013.952,-97.895,389.553,-23.988,21.670,-44.241
C06954=1013.948,-98.215,389.576,-23.987,21.670,-44.246
C06955=1013.945,-98.536,389.599,-23.987,21.672,-44.250
C06956=1013.940,-98.857,389.623,-23.986,21.671,-44.255
C06957=1013.937,-99.179,389.646,-23.986,21.673,-44.260
C06958=1013.932,-99.500,389.670,-23.985,21.673,-44.265
C06959=1013.917,-100.647,389.754,-24.004,21.745,-44.237
C06960=1013.912,-101.047,389.783,-24.042,21.880,-44.155
C06961=1013.907,-101.429,389.811,-24.079,22.010,-44.078
C06962=1013.903,-101.812,389.839,-24.117,22.142,-44.000
C06963=1013.898,-102.196,389.867,-24.154,22.274,-43.922
C06964=1013.892,-102.580,389.895,-24.191,22.407,-43.844
C06965=1013.888,-102.965,389.924,-24.228,22.541,-43.766
C06966=1013.883,-103.351,389.951,-24.266,22.677,-43.687
C06967=1013.877,-103.737,389.980,-24.303,22.814,-43.609
C06968=1013.872,-104.124,390.008,-24.341,22.953,-43.528
C06969=1013.866,-104.511,390.037,-24.379,23.091,-43.450
C06970=1013.862,-104.899,390.065,-24.416,23.231,-43.370
C06971=1013.856,-105.287,390.093,-24.454,23.373,-43.290
C06972=1013.851,-105.676,390.122,-24.492,23.515,-43.209
C06973=1013.846,-106.065,390.151,-24.530,23.659,-43.129
C06974=1013.840,-106.455,390.179,-24.568,23.804,-43.048
C06975=1013.834,-106.863,390.208,-24.608,23.956,-42.965
C06976=1013.832,-107.077,390.224,-24.629,24.036,-42.921
C06977=1013.829,-107.297,390.240,-24.650,24.119,-42.875
C06978=1013.826,-107.524,390.257,-24.673,24.205,-42.827
C06979=1013.822,-107.753,390.274,-24.695,24.293,-42.778
C06980=1013.819,-107.986,390.291,-24.718,24.381,-42.729
C06981=1013.816,-108.218,390.308,-24.740,24.470,-42.681
C06982=1013.813,-108.447,390.325,-24.763,24.558,-42.633
C06983=1013.809,-108.672,390.341,-24.785,24.644,-42.585
C06984=1013.806,-108.891,390.358,-24.806,24.729,-42.539
C06985=1013.799,-109.308,390.388,-24.847,24.891,-42.453
C06986=1013.795,-109.702,390.417,-24.885,25.045,-42.371
C06987=1013.788,-110.091,390.445,-24.923,25.198,-42.290
C06988=1013.783,-110.480,390.474,-24.961,25.351,-42.208
C06989=1013.777,-110.869,390.502,-24.999,25.507,-42.127
C06990=1013.772,-111.258,390.530,-25.036,25.663,-42.045
C06991=1013.766,-111.645,390.559,-25.074,25.820,-41.964
C06992=1013.761,-112.035,390.588,-25.112,25.977,-41.882
C06993=1013.755,-112.423,390.616,-25.149,26.136,-41.801
C06994=1013.749,-112.812,390.645,-25.187,26.294,-41.720
C06995=1013.744,-113.200,390.673,-25.224,26.455,-41.638
C06996=1013.737,-113.589,390.701,-25.262,26.617,-41.555
C06997=1013.732,-113.977,390.730,-25.299,26.778,-41.474
C06998=1013.726,-114.366,390.759,-25.337,26.941,-41.393
C06999=1013.720,-114.754,390.787,-25.374,27.106,-41.310
C07000=1013.714,-115.143,390.815,-25.412,27.270,-41.230
C07001=1013.708,-115.531,390.845,-25.449,27.437,-41.147
C07002=1013.703,-115.919,390.872,-25.486,27.603,-41.066
C07003=1013.696,-116.308,390.901,-25.523,27.771,-40.984
C07004=1013.690,-116.695,390.930,-25.560,27.939,-40.903
C07005=1013.685,-117.085,390.959,-25.598,28.109,-40.821
C07006=1013.679,-117.472,390.987,-25.634,28.279,-40.739
C07007=1013.672,-117.861,391.016,-25.671,28.450,-40.658
C07008=1013.667,-118.249,391.044,-25.708,28.622,-40.577
C07009=1013.661,-118.637,391.073,-25.745,28.795,-40.496
C07010=1013.654,-119.026,391.101,-25.781,28.969,-40.414
C07011=1013.648,-119.414,391.130,-25.818,29.143,-40.334
C07012=1013.642,-119.802,391.158,-25.854,29.319,-40.253
C07013=1013.636,-120.190,391.187,-25.891,29.496,-40.171
C07014=1013.629,-120.578,391.216,-25.927,29.673,-40.091
C07015=1013.624,-120.966,391.244,-25.963,29.852,-40.008
C07016=1013.618,-121.354,391.272,-25.999,30.031,-39.929
C07017=1013.611,-121.743,391.301,-26.035,30.211,-39.847
C07018=1013.605,-122.130,391.330,-26.071,30.392,-39.767
C07019=1013.598,-122.519,391.359,-26.107,30.573,-39.687
C07020=1013.593,-122.906,391.387,-26.143,30.757,-39.607
C07021=1013.586,-123.295,391.416,-26.178,30.940,-39.526
C07022=1013.580,-123.683,391.445,-26.214,31.125,-39.447
C07023=1013.573,-124.071,391.474,-26.249,31.310,-39.366
C07024=1013.567,-124.459,391.502,-26.285,31.496,-39.287
C07025=1013.562,-124.846,391.531,-26.320,31.683,-39.208
C07026=1013.555,-125.235,391.560,-26.355,31.871,-39.128
C07027=1013.549,-125.622,391.589,-26.390,32.060,-39.049
C07028=1013.542,-126.011,391.617,-26.425,32.249,-38.970
C07029=1013.536,-126.399,391.646,-26.460,32.440,-38.890
C07030=1013.530,-126.787,391.675,-26.494,32.631,-38.813
C07031=1013.524,-127.175,391.704,-26.529,32.824,-38.733
C07032=1013.518,-127.546,391.731,-26.562,33.009,-38.658
C07033=1013.511,-127.950,391.760,-26.598,33.211,-38.577
C07034=1013.505,-128.338,391.789,-26.632,33.405,-38.499
C07035=1013.498,-128.726,391.819,-26.666,33.602,-38.421
C07036=1013.492,-129.114,391.847,-26.700,33.797,-38.344
C07037=1013.485,-129.502,391.876,-26.734,33.995,-38.267
C07038=1013.479,-129.890,391.905,-26.767,34.194,-38.189
C07039=1013.472,-130.278,391.934,-26.801,34.393,-38.111
C07040=1013.466,-130.665,391.962,-26.834,34.591,-38.036
C07041=1013.459,-131.053,391.991,-26.868,34.793,-37.958
C07042=1013.453,-131.441,392.020,-26.901,34.994,-37.883
C07043=1013.446,-131.829,392.050,-26.934,35.196,-37.806
C07044=1013.440,-132.217,392.078,-26.967,35.399,-37.731
C07045=1013.434,-132.604,392.107,-27.000,35.601,-37.655
C07046=1013.427,-132.992,392.136,-27.032,35.805,-37.581
C07047=1013.421,-133.379,392.164,-27.065,36.011,-37.506
C07048=1013.414,-133.767,392.194,-27.097,36.216,-37.431
C07049=1013.408,-134.155,392.223,-27.129,36.422,-37.356
C07050=1013.834,-134.175,391.879,-24.572,24.018,-43.329
C07051=1013.838,-133.981,391.865,-24.544,23.911,-43.391
C07052=1013.846,-133.594,391.837,-24.486,23.697,-43.515
C07053=1013.854,-133.206,391.810,-24.428,23.483,-43.640
C07054=1013.862,-132.818,391.782,-24.370,23.270,-43.764
C07055=1013.870,-132.430,391.754,-24.311,23.059,-43.890
C07056=1013.877,-132.042,391.726,-24.252,22.848,-44.015
C07057=1013.885,-131.654,391.698,-24.193,22.637,-44.143
C07058=1013.893,-131.267,391.670,-24.133,22.428,-44.269
C07059=1013.901,-130.879,391.642,-24.073,22.220,-44.397
C07060=1013.909,-130.491,391.615,-24.013,22.014,-44.524
C07061=1013.916,-130.123,391.587,-23.956,21.818,-44.646
C07062=1013.939,-128.976,391.505,-23.930,21.723,-44.689
C07063=1013.945,-128.648,391.482,-23.931,21.723,-44.686
C07064=1013.952,-128.320,391.459,-23.931,21.722,-44.680
C07065=1013.959,-127.991,391.435,-23.932,21.721,-44.676
C07066=1013.965,-127.663,391.412,-23.933,21.721,-44.671
C07067=1013.972,-127.335,391.388,-23.933,21.720,-44.667
C07068=1013.978,-127.007,391.364,-23.934,21.720,-44.662
C07069=1013.984,-126.678,391.341,-23.935,21.720,-44.657
C07070=1013.990,-126.350,391.318,-23.935,21.719,-44.652
C07071=1013.996,-126.022,391.293,-23.936,21.719,-44.647
C07072=1014.002,-125.693,391.270,-23.936,21.717,-44.643
C07073=1014.008,-125.365,391.247,-23.937,21.717,-44.638
C07074=1014.015,-125.037,391.223,-23.937,21.717,-44.634
C07075=1014.021,-124.708,391.200,-23.938,21.716,-44.628
C07076=1014.027,-124.380,391.177,-23.939,21.715,-44.625
C07077=1014.032,-124.052,391.153,-23.939,21.715,-44.620
C07078=1014.038,-123.723,391.130,-23.940,21.714,-44.615
C07079=1014.044,-123.395,391.106,-23.940,21.714,-44.610
C07080=1014.050,-123.067,391.082,-23.941,21.713,-44.606
C07081=1014.056,-122.738,391.059,-23.942,21.713,-44.601
C07082=1014.062,-122.410,391.035,-23.942,21.712,-44.597
C07083=1014.067,-122.082,391.012,-23.943,21.711,-44.591
C07084=1014.073,-121.754,390.988,-23.944,21.711,-44.586
C07085=1014.079,-121.424,390.965,-23.944,21.710,-44.582
C07086=1014.085,-121.096,390.941,-23.945,21.710,-44.577
C07087=1014.090,-120.767,390.918,-23.945,21.709,-44.573
C07088=1014.096,-120.440,390.894,-23.946,21.709,-44.568
C07089=1014.101,-120.111,390.871,-23.946,21.708,-44.564
C07090=1014.107,-119.782,390.847,-23.947,21.707,-44.558
C07091=1014.113,-119.454,390.823,-23.948,21.707,-44.554
C07092=1014.118,-119.125,390.800,-23.948,21.707,-44.549
C07093=1014.123,-118.797,390.776,-23.949,21.705,-44.545
C07094=1014.129,-118.468,390.753,-23.949,21.705,-44.540
C07095=1014.134,-118.140,390.730,-23.950,21.705,-44.535
C07096=1014.139,-117.811,390.706,-23.951,21.704,-44.531
C07097=1014.145,-117.482,390.682,-23.951,21.704,-44.525
C07098=1014.149,-117.154,390.659,-23.952,21.703,-44.521
C07099=1014.155,-116.825,390.635,-23.953,21.703,-44.516
C07100=1014.160,-116.497,390.611,-23.953,21.701,-44.512
C07101=1014.165,-116.168,390.588,-23.954,21.701,-44.507
C07102=1014.170,-115.839,390.564,-23.954,21.701,-44.503
C07103=1014.175,-115.510,390.541,-23.955,21.700,-44.497
C07104=1014.180,-115.182,390.517,-23.956,21.700,-44.492
C07105=1014.186,-114.853,390.493,-23.956,21.699,-44.488
C07106=1014.191,-114.524,390.470,-23.957,21.699,-44.483
C07107=1014.196,-114.196,390.447,-23.957,21.698,-44.479
C07108=1014.201,-113.867,390.423,-23.958,21.697,-44.473
C07109=1014.206,-113.539,390.400,-23.958,21.697,-44.470
C07110=1014.210,-113.209,390.376,-23.959,21.696,-44.464
C07111=1014.216,-112.880,390.352,-23.960,21.696,-44.459
C07112=1014.220,-112.552,390.328,-23.960,21.695,-44.455
C07113=1014.225,-112.223,390.304,-23.961,21.695,-44.449
C07114=1014.230,-111.895,390.281,-23.962,21.694,-44.446
C07115=1014.235,-111.566,390.257,-23.962,21.693,-44.440
C07116=1014.239,-111.237,390.234,-23.963,21.693,-44.436
C07117=1014.244,-110.908,390.210,-23.963,21.692,-44.431
C07118=1014.249,-110.579,390.186,-23.964,21.692,-44.426
C07119=1014.253,-110.250,390.163,-23.965,21.691,-44.422
C07120=1014.258,-109.920,390.139,-23.965,21.691,-44.416
C07121=1014.262,-109.592,390.116,-23.966,21.690,-44.412
C07122=1014.267,-109.263,390.092,-23.967,21.689,-44.407
C07123=1014.271,-108.934,390.068,-23.967,21.689,-44.402
C07124=1014.276,-108.605,390.045,-23.968,21.689,-44.398
C07125=1014.281,-108.276,390.020,-23.969,21.688,-44.392
C07126=1014.285,-107.947,389.997,-23.969,21.687,-44.388
C07127=1014.290,-107.617,389.974,-23.970,21.687,-44.383
C07128=1014.294,-107.289,389.950,-23.971,21.687,-44.378
C07129=1014.298,-106.959,389.926,-23.971,21.685,-44.374
C07130=1014.302,-106.631,389.902,-23.972,21.685,-44.368
C07131=1014.307,-106.301,389.878,-23.972,21.685,-44.365
C07132=1014.311,-105.972,389.856,-23.973,21.684,-44.359
C07133=1014.315,-105.644,389.832,-23.974,21.684,-44.354
C07134=1014.319,-105.314,389.808,-23.974,21.683,-44.350
C07135=1014.323,-104.987,389.784,-23.975,21.683,-44.344
C07136=1014.328,-104.659,389.760,-23.975,21.681,-44.340
C07137=1014.332,-104.330,389.737,-23.976,21.681,-44.335
C07138=1014.336,-104.003,389.713,-23.976,21.681,-44.331
C07139=1014.340,-103.676,389.689,-23.977,21.680,-44.326
C07140=1014.343,-103.349,389.666,-23.978,21.680,-44.320
C07141=1014.348,-103.024,389.642,-23.978,21.679,-44.316
C07142=1014.351,-102.697,389.619,-23.979,21.679,-44.311
C07143=1014.355,-102.372,389.595,-23.980,21.678,-44.307
C07144=1014.359,-102.048,389.572,-23.980,21.677,-44.302
C07145=1014.363,-101.723,389.548,-23.981,21.677,-44.298
C07146=1014.367,-101.400,389.525,-23.981,21.676,-44.292
C07147=1014.371,-101.077,389.501,-23.982,21.676,-44.287
C07148=1014.374,-100.754,389.479,-23.983,21.675,-44.283
C07149=1014.378,-100.432,389.455,-23.983,21.675,-44.278
C07150=1014.382,-100.110,389.431,-23.984,21.674,-44.274
C07151=1014.385,-99.788,389.408,-23.985,21.673,-44.268
C07152=1014.390,-99.467,389.385,-23.985,21.673,-44.265
C07153=1014.393,-99.146,389.361,-23.986,21.673,-44.260
C07154=1014.396,-98.825,389.339,-23.986,21.671,-44.255
C07155=1014.400,-98.504,389.315,-23.987,21.672,-44.250
C07156=1014.404,-98.183,389.292,-23.987,21.670,-44.246
C07157=1014.407,-97.861,389.269,-23.988,21.670,-44.241
C07158=1014.411,-97.541,389.245,-23.989,21.670,-44.236
C07159=1014.414,-97.220,389.222,-23.989,21.669,-44.231
C07160=1014.417,-96.898,389.199,-23.990,21.669,-44.226
C07161=1014.420,-96.577,389.175,-23.991,21.668,-44.222
C07162=1014.424,-96.255,389.152,-23.991,21.668,-44.217
C07163=1014.428,-95.933,389.128,-23.992,21.667,-44.213
C07164=1014.431,-95.611,389.105,-23.993,21.666,-44.207
C07165=1014.434,-95.288,389.081,-23.993,21.666,-44.204
C07166=1014.438,-94.965,389.058,-23.994,21.666,-44.199
C07167=1014.441,-94.641,389.035,-23.994,21.665,-44.193
C07168=1014.444,-94.317,389.011,-23.995,21.664,-44.189
C07169=1014.448,-93.992,388.987,-23.996,21.664,-44.184
C07170=1014.450,-93.667,388.963,-23.996,21.663,-44.180
C07171=1014.454,-93.342,388.940,-23.997,21.663,-44.175
C07172=1014.457,-93.015,388.916,-23.998,21.662,-44.169
C07173=1014.460,-92.689,388.892,-23.998,21.662,-44.165
C07174=1014.463,-92.361,388.869,-23.999,21.661,-44.160
C07175=1014.466,-92.033,388.844,-23.999,21.660,-44.156
C07176=1014.470,-91.705,388.821,-24.000,21.660,-44.150
C07177=1014.473,-91.376,388.796,-24.001,21.660,-44.145
C07178=1014.476,-91.047,388.773,-24.001,21.659,-44.141
C07179=1014.479,-90.717,388.749,-24.002,21.658,-44.136
C07180=1014.482,-90.379,388.724,-24.003,21.658,-44.130
C07181=1014.486,-89.973,388.695,-24.004,21.657,-44.123
C07182=1014.488,-89.742,388.677,-24.004,21.656,-44.121
C07183=1014.490,-89.504,388.660,-24.004,21.656,-44.119
C07184=1014.492,-89.270,388.643,-24.004,21.656,-44.117
C07185=1014.493,-89.050,388.627,-24.005,21.656,-44.114
C07186=1014.497,-88.680,388.600,-24.006,21.655,-44.106
C07187=1014.500,-88.361,388.576,-24.006,21.654,-44.102
C07188=1014.503,-88.048,388.553,-24.007,21.654,-44.097
C07189=1014.505,-87.738,388.530,-24.007,21.653,-44.093
C07190=1014.508,-87.425,388.508,-24.008,21.653,-44.088
C07191=1014.510,-87.109,388.485,-24.009,21.652,-44.082
C07192=1014.513,-86.786,388.461,-24.009,21.652,-44.078
C07193=1014.516,-86.457,388.437,-24.010,21.651,-44.073
C07194=1014.519,-86.098,388.411,-24.011,21.650,-44.067
C07195=1014.522,-85.689,388.380,-24.012,21.649,-44.062
C07196=1014.524,-85.475,388.365,-24.012,21.649,-44.060
C07197=1014.526,-85.263,388.349,-24.012,21.650,-44.056
C07198=1014.528,-84.865,388.320,-24.013,21.649,-44.051
C07199=1014.531,-84.516,388.295,-24.014,21.648,-44.045
C07200=1014.535,-84.182,388.270,-24.015,21.648,-44.040
C07201=1014.537,-83.846,388.245,-24.015,21.647,-44.036
C07202=1014.539,-83.511,388.220,-24.016,21.647,-44.031
C07203=1014.542,-83.175,388.196,-24.016,21.646,-44.025
C07204=1014.544,-82.839,388.172,-24.017,21.645,-44.021
C07205=1014.548,-82.503,388.146,-24.018,21.645,-44.016
C07206=1014.549,-82.166,388.121,-24.018,21.645,-44.010
C07207=1014.552,-81.829,388.097,-24.019,21.644,-44.005
C07208=1014.554,-81.490,388.072,-24.020,21.643,-44.001
C07209=1014.557,-81.153,388.046,-24.020,21.643,-43.995
C07210=1014.559,-80.814,388.021,-24.021,21.643,-43.990
C07211=1014.562,-80.474,387.997,-24.021,21.641,-43.986
C07212=1014.564,-80.135,387.972,-24.022,21.641,-43.981
C07213=1014.566,-79.796,387.946,-24.023,21.641,-43.975
C07214=1014.569,-79.455,387.922,-24.023,21.639,-43.971
C07215=1014.571,-79.115,387.897,-24.024,21.639,-43.966
C07216=1014.573,-78.774,387.871,-24.025,21.638,-43.960
C07217=1014.576,-78.432,387.846,-24.026,21.639,-43.955
C07218=1014.578,-78.091,387.821,-24.026,21.637,-43.951
C07219=1014.579,-77.749,387.796,-24.027,21.637,-43.946
C07220=1014.582,-77.407,387.771,-24.028,21.636,-43.940
C07221=1014.584,-77.064,387.745,-24.028,21.636,-43.936
C07222=1014.587,-76.722,387.720,-24.029,21.635,-43.931
C07223=1014.588,-76.380,387.694,-24.030,21.635,-43.926
C07224=1014.591,-76.037,387.668,-24.030,21.634,-43.920
C07225=1014.593,-75.693,387.643,-24.031,21.634,-43.916
C07226=1014.595,-75.350,387.617,-24.031,21.633,-43.911
C07227=1014.597,-75.007,387.592,-24.032,21.633,-43.905
C07228=1014.599,-74.663,387.567,-24.033,21.632,-43.901
C07229=1014.601,-74.320,387.541,-24.033,21.632,-43.896
C07230=1014.603,-73.977,387.516,-24.034,21.631,-43.890
C07231=1014.604,-73.633,387.490,-24.035,21.630,-43.885
C07232=1014.607,-73.288,387.465,-24.035,21.630,-43.881
C07233=1014.608,-72.944,387.439,-24.036,21.629,-43.875
C07234=1014.610,-72.601,387.414,-24.037,21.629,-43.870
C07235=1014.612,-72.256,387.388,-24.038,21.628,-43.865
C07236=1014.614,-71.912,387.362,-24.038,21.628,-43.861
C07237=1014.616,-71.568,387.336,-24.039,21.627,-43.855
C07238=1014.618,-71.224,387.311,-24.040,21.627,-43.850
C07239=1014.619,-70.880,387.285,-24.040,21.626,-43.844
C07240=1014.622,-70.536,387.260,-24.041,21.625,-43.840
C07241=1014.623,-70.192,387.234,-24.041,21.625,-43.835
C07242=1014.624,-69.848,387.208,-24.042,21.624,-43.829
C07243=1014.627,-69.504,387.183,-24.043,21.624,-43.824
C07244=1014.628,-69.160,387.157,-24.043,21.623,-43.820
C07245=1014.629,-68.816,387.131,-24.044,21.623,-43.815
C07246=1014.632,-68.473,387.105,-24.045,21.622,-43.809
C07247=1014.633,-68.129,387.080,-24.045,21.622,-43.805
C07248=1014.634,-67.785,387.054,-24.046,21.621,-43.800
C07249=1014.636,-67.442,387.028,-24.047,21.621,-43.795
C07250=1014.637,-67.099,387.002,-24.048,21.620,-43.789
C07251=1014.639,-66.756,386.977,-24.048,21.620,-43.785
C07252=1014.640,-66.412,386.951,-24.049,21.619,-43.780
C07253=1014.642,-66.070,386.926,-24.050,21.619,-43.774
C07254=1014.643,-65.728,386.900,-24.050,21.617,-43.770
C07255=1014.644,-65.385,386.874,-24.051,21.618,-43.765
C07256=1014.646,-65.044,386.848,-24.051,21.617,-43.759
C07257=1014.648,-64.702,386.823,-24.052,21.617,-43.754
C07258=1014.649,-64.361,386.797,-24.053,21.615,-43.750
C07259=1014.650,-64.019,386.772,-24.053,21.616,-43.745
C07260=1014.651,-63.679,386.746,-24.054,21.615,-43.739
C07261=1014.653,-63.339,386.720,-24.055,21.614,-43.735
C07262=1014.654,-62.999,386.695,-24.055,21.613,-43.730
C07263=1014.655,-62.659,386.668,-24.056,21.614,-43.725
C07264=1014.656,-62.320,386.644,-24.057,21.612,-43.720
C07265=1014.657,-61.981,386.618,-24.057,21.612,-43.715
C07266=1014.658,-61.643,386.592,-24.058,21.611,-43.710
C07267=1014.659,-61.305,386.567,-24.059,21.611,-43.706
C07268=1014.660,-60.967,386.541,-24.059,21.610,-43.700
C07269=1014.661,-60.630,386.516,-24.060,21.610,-43.695
C07270=1014.663,-60.293,386.491,-24.060,21.609,-43.691
C07271=1014.663,-59.957,386.465,-24.061,21.609,-43.686
C07272=1014.665,-59.621,386.440,-24.062,21.608,-43.680
C07273=1014.666,-59.285,386.414,-24.062,21.608,-43.676
C07274=1014.667,-58.950,386.389,-24.063,21.607,-43.671
C07275=1014.668,-58.615,386.364,-24.064,21.607,-43.666
C07276=1014.669,-58.280,386.339,-24.064,21.606,-43.662
C07277=1014.670,-57.946,386.313,-24.065,21.606,-43.656
C07278=1014.670,-57.612,386.288,-24.066,21.605,-43.652
C07279=1014.671,-57.278,386.262,-24.066,21.604,-43.647
C07280=1014.673,-56.945,386.237,-24.067,21.605,-43.642
